# B&R Automation Studio project Y4_V3_1 (part 2)

### Acp10cfg.ncc - 5PPC2100_BY01_000/Motion/Acp10cfg.ncc
```
NcConfiguration (Version=2.46.0, NcSwId=Acp10)
  ACP10CF1_typ:
    cnt_nettrc_rec_drive = 150
    bufsize_trace_upload = 1200
    tc_nc_man_task = Cyclic #1
    glob_pv_as_ncobject = Yes
    ncsys_dl_broadcast = Yes
    ncsys_dl_acp_reset = Yes
    safemc_log_err_to_ax = Yes
    network_init:
      ncsw_init_execute = Yes
      automatic_execute = No
      node_nr_warning = Yes
      net_err_before_ncact = Yes
    nettrc:
      enter_parsecrec = Yes
      enter_ncaction = Yes
      save_ring_startidx = Yes
    cam_prof_download:
      cam_dat_dl_parallel = No
      tc_cam_dl_parallel = Task class for NC Manager task
    plk_if[0]:
      if_name = SL1.IF1
      tc_CycDat_PLCopen = Task class for NC Manager task
      mc_broadcast_extdat = No
    plk_if[1]:
      if_name = SS1.SS1.SS1.SS1.SS1
      tc_CycDat_PLCopen = Task class for NC Manager task
      mc_broadcast_extdat = No
    sdc_if[0]:
      if_name = SDC_IF1
      mc_broadcast_size = 800
      mc_broadcast_extdat = No
```

### Acp10map.ncm - 5PPC2100_BY01_000/Motion/Acp10map.ncm
```
NcMapping (NcSwId=Acp10, DisabledNodesAreHidden=False)
  NcObject Axis1 (ModuleId=8V1045.00-2a, Type=ncAXIS, Channel=1, AcoposSimulation=Off, InitParameter=axis1, AcoposParameter=table_par1, Disabled=FALSE, ModuleDisabled=FALSE)
  NcObject 8V1045.00-2a_ncV_AXIS1 (ModuleId=8V1045.00-2a, Type=ncV_AXIS, Channel=1, Disabled=TRUE, ModuleDisabled=FALSE)
  NcObject Axis2 (ModuleId=8V1045.00-2, Type=ncAXIS, Channel=1, AcoposSimulation=Off, InitParameter=axis1, AcoposParameter=table_par1, Disabled=FALSE, ModuleDisabled=FALSE)
  NcObject 8V1045.00-2_ncV_AXIS1 (ModuleId=8V1045.00-2, Type=ncV_AXIS, Channel=1, Disabled=TRUE, ModuleDisabled=FALSE)
  NcObject 8I74xxxxxxx.01P-1_ncAXIS1 (ModuleId=INV2, Type=ncAXIS, Channel=1, AcoposSimulation=Off, Disabled=TRUE, ModuleDisabled=FALSE)
  NcObject 8I74xxxxxxx.01P-1_ncAXIS1 (ModuleId=INV7, Type=ncAXIS, Channel=1, AcoposSimulation=Off, Disabled=TRUE, ModuleDisabled=FALSE)
  NcObject 8I74xxxxxxx.01P-1_ncAXIS1 (ModuleId=INV10, Type=ncAXIS, Channel=1, AcoposSimulation=Off, Disabled=TRUE, ModuleDisabled=FALSE)
  NcObject 8I74xxxxxxx.01P-1_ncAXIS1 (ModuleId=INV13, Type=ncAXIS, Channel=1, AcoposSimulation=Off, Disabled=TRUE, ModuleDisabled=FALSE)
  NcObject 8I74xxxxxxx.01P-1_ncAXIS1 (ModuleId=INV11, Type=ncAXIS, Channel=1, AcoposSimulation=Off, Disabled=TRUE, ModuleDisabled=FALSE)
  NcObject 8I74xxxxxxx.01P-1_ncAXIS1 (ModuleId=INV12, Type=ncAXIS, Channel=1, AcoposSimulation=Off, Disabled=TRUE, ModuleDisabled=FALSE)
```

## Configuration Simulation

CPU , AutomationRuntime D4.24, Vc V4.26.0

### Task classes (Cpu.sw)
```
Cyclic#1 (cycle 500 us, tolerance 100000 us):
  IO <- System.IO.prg
  LineConfig <- System.LineConfig.prg
  SensorInpu <- System.SensorInput.prg
  Seam1Array <- Motion.Seam1Array.prg
  Seam2Array <- Motion.Seam2Array.prg
Cyclic#2 (cycle 200000 us, tolerance 10000000 us):
  ResetInv <- Automatic.ResetInv.prg
  AxBlocks <- Automatic.AxBlocks.prg
  ConLoad <- Automatic.ConLoad.prg
  ConSeam1 <- Automatic.ConSeam1.prg
  ConCorner <- Automatic.ConCorner.prg
  ConSeam2 <- Automatic.ConSeam2.prg
  ConBuffers <- Automatic.ConBuffers.prg
  ConRow <- Automatic.ConRow.prg
  ConBatch <- Automatic.ConBatch.prg
  Seaming <- Automatic.Seaming.prg
  Batching <- Automatic.Batching.prg
  Modes <- Automatic.Modes.prg
  FlipUpArms <- Automatic.FlipUpArms.prg
  Outputs <- Automatic.Outputs.prg
Cyclic#3 (cycle 500000 us, tolerance 10000000 us):
  Control <- System.Control.prg
  Seamers <- System.Seamers.prg
  Process <- System.Process.prg
Cyclic#4 (cycle 1000000 us, tolerance 10000000 us):
  IPConfig <- IPConfig.IPConfig.prg
  Filstar <- System.Filstar.prg
  Level <- VisControl.HMIControl.Level.prg
  Status <- VisControl.HMIControl.Status.prg
  Start <- VisControl.HMIControl.Start.prg
  ESRecover <- VisControl.HMIControl.ESRecover.prg
  Simulation <- VisControl.HMIControl.Simulation.prg
  Page10 <- VisControl.HMIControl.Page10.prg
  Page11 <- VisControl.HMIControl.Page11.prg
  Page12 <- VisControl.HMIControl.Page12.prg
  Page13 <- VisControl.HMIControl.Page13.prg
  Page14 <- VisControl.HMIControl.Page14.prg
  Page15 <- VisControl.HMIControl.Page15.prg
  Page16 <- VisControl.HMIControl.Page16.prg
  Page17 <- VisControl.HMIControl.Page17.prg
  Page18 <- VisControl.HMIControl.Page18.prg
  Page20 <- VisControl.HMIControl.Page20.prg
  EPLComms <- InvComms.EPLComms.prg
  BatchData <- VisControl.BatchDisp.BatchData.prg
VcDataObjects: HMIXGA <- HMIXGA.HMIXGA.dob, BatchP <- BatchDisplay.BatchP.dob
Binaries: verdana, vcpkat, vctcal, HMIXGA03, vcgclass, vcnet, HMIXGA01, vcpdsw, vccshape, arialbd, arialn, vccstr, trebuc, vccnum, vcrt, visvc, vccbar, vcbclass, vcalarm, vcctext, vcmgr, vccovl, HMIXGA02, vccalarm, vcpfar00, vcdsloc, vccbtn, vcdsint, vcchspot, arial, vccpwd, vcfile, vcpdvnc, vcshared, vccbmp, vcfntttf, vccddbox, vccpopup, SRVXGA01, SRVXGA02, SRVXGA03, SRVXGA, BatchP01, BatchP03, BatchP02, acp10cfg, Acp10map, ashwd, arconfig, asfw, sysconf, iomap, Acp10sys, vcchtml, vccurl, vcxml, vccdt, VisuTe01, VisuTe02, VisuTe03, vcctrend, vccslider, vccline
Libraries: AsIecCon, astime, standard, sys_lib, Runtime, brsystem, powerlnk, DataObj, asstring, dvframe, AxisCtrl, AsARCfg, IecCheck, LoopConR, Visapi, vcresman, Acp10man, Acp10par, NcGlobal, fileio, Acp10_MC, Lib_Ashton, asepl, AsMath, arsvcreg
```

### Hardware
```
PC_any : PC_any v1.1.0.0 (OrderNumber=PC)
  Connector IF3:
    Vnc1
    VncVcObjectName1 = HMIXGA
    VncKeyMappingFile1 = VC\PS2-Keyboard.dis
    VncAuthentication1 = 1
    VncPasswordViewOnly1 = 1234
    VncPasswordViewControl1 = 4046
    VncRefreshRate1 = 100
    Vnc2
    VncVcObjectName2 = BatchP
    VncKeyMappingFile2 = VC\PS2-Keyboard1.dis
    VncPortNumber2 = 5902
  ConfigurationID = N13_V1_0_Simulation
  PermanentPvSize = 4096
  VolatileGlobalPvSize = 327679
  CyclicObjects = 250
  BRObjects = 600
  SystemTick = 500
  Cyclic1Duration = 500
  Cyclic1Tolerance = 100000
  Cyclic1Input = 1
  Cyclic2Duration = 200000
  Cyclic2Tolerance = 10000000
  Cyclic3Duration = 500000
  Cyclic3Tolerance = 10000000
  Cyclic4Duration = 1000000
  Cyclic4Tolerance = 10000000
  Cyclic5Duration = 2000000
  Cyclic5Tolerance = 10000000
  Cyclic6Duration = 3000000
  Cyclic6Tolerance = 12000000
  Cyclic7Duration = 4000000
  Cyclic7Tolerance = 12000000
  Cyclic8Duration = 5000000
  Cyclic8Tolerance = 30000000
```

### Cpu.per - PC_any/Cpu.per
```iecst
(********************************************************************
 * COPYRIGHT --
 ********************************************************************
 * File: Cpu.per
 * Author: NickE
 * Created: April 2, 2015
 ********************************************************************
 * Declaration of permanent variables
 ********************************************************************)
VAR_CONFIG
	Ax1P AT %M0; (*Axis 1 permananent variables*)
	Ax2P AT %M60; (*Axis 2 permananent variables*)
	Grind1 AT %M120; (*Grinding data permanent variables*)
	Grind2 AT %M176; (*Grinding data permanent variables*)
	Data AT %M232; (*Runtime data permanent variables*)
	PresetSys AT %M264; (*System timer presets*)
	SysPerm AT %M344; (*Permanent system variables*)
	PresetSeam AT %M368; (*Auto running timer presets*)
	RowPerm AT %M472; (*Row building permanent variables*)
	LoadPerm AT %M488; (*Load building permanent variables*)
	ArmsPerm1 AT %M504; (*Flip up arms retained values*)
	ArmsPerm2 AT %M528; (*Flip up arms retained values*)
	ScalePerm AT %M552; (*Conveyor scaling constants*)
	InvPerms AT %M608; (*Inverter Permanent Variables*)
	Speeds AT %M724; (*Conveyor speeds*)
	AnalogPerm AT %M768; (* *)
	TrackDelayPT AT %M1104; (*Preset for timeout*)
	NozzlePerm AT %M1364; (* *)
	InterceptPT AT %M1372; (* *)
END_VAR
```

### Acp10cfg.ncc - PC_any/Motion/Acp10cfg.ncc
```
NcConfiguration (Version=2.45.1, NcSwId=Acp10)
  ACP10CF1_typ:
    cnt_nettrc_rec_drive = 150
    bufsize_trace_upload = 1200
    tc_nc_man_task = Cyclic #1
    glob_pv_as_ncobject = Yes
    ncsys_dl_broadcast = Yes
    ncsys_dl_acp_reset = Yes
    safemc_log_err_to_ax = Yes
    network_init:
      ncsw_init_execute = Yes
      automatic_execute = No
      node_nr_warning = Yes
      net_err_before_ncact = Yes
    nettrc:
      enter_parsecrec = Yes
      enter_ncaction = Yes
      save_ring_startidx = No
    cam_prof_download:
      cam_dat_dl_parallel = No
      tc_cam_dl_parallel = Task class for NC Manager task
```

## Logical view

Binary libraries used (declarations not repeated): Runtime, Operator, standard, sys_lib, brsystem, powerlnk, AsIecCon, astime, DataObj, asstring, dvframe, AsARCfg, LoopConR 2.72.0, Visapi, AsEPL, AsMath, Acp10man 2.50.1, Acp10par 2.50.1, NcGlobal 2.50.1, Acp10_MC 2.50.1

### Global.typ - Global data types
```iecst
(********************************************************************
 * COPYRIGHT --
 ********************************************************************
 * File: Global.typ
 * Author: NickE
 * Created: April 2, 2015
 ********************************************************************
 * Global data types of project N_Default
 ********************************************************************)

TYPE
	SizeData_enum :
		(
		SD_Idle := 0, (*Wait*)
		SD_WidthData := 1, (*Set Width Data*)
		SD_WidthACK := 2, (*Wait for acknowledgement that width data has been received*)
		SD_NotWidthACK := 3, (*Wait for acknowledge off, data has transmitted*)
		SD_LengthData := 4, (*Set Length Data*)
		SD_LengthACK := 5, (*Wait for acknowledgement that length data has been received*)
		SD_NotLengthACK := 6 (*Wait for acknowledge off, data has transmitted*)
		);
	SizeData_typ : 	STRUCT
		Sizes : ARRAY[0..11]OF BOOL; (*Bit array to pass data to AGV controller*)
		Sequence : SizeData_enum;
		CurrentWidth : UINT;
		CurrentLength : UINT;
		WidthMask : BOOL;
		LengthMask : BOOL;
	END_STRUCT;
	Measurement_typ : 	STRUCT
		Reset : BOOL;
		Runtime : Display_enum;
	END_STRUCT;
	Alarm_typ : 	STRUCT
		Control : USINT; (*Visu alarm control*)
		Group : USINT; (*Visu alarm control*)
		Alarm : USINT; (*Visu alarm control*)
		Priority : USINT; (*Visu alarm control*)
	END_STRUCT;
	ANALOGCAPTURE_typ : 	STRUCT
		CLB : ANALOGRECORD_typ;
	END_STRUCT;
	ANALOGPERMS_typ : 	STRUCT
		V1 : ANALOGPERM_typ;
		C1 : ANALOGPERM_typ;
		C2 : ANALOGPERM_typ;
	END_STRUCT;
	ANALOGPERM_typ : 	STRUCT
		ActAnalog : REAL;
		ActSpeed : REAL;
	END_STRUCT;
	ANALOGRECORD_typ : 	STRUCT
		RecordStart : BOOL;
		RecordConfirm : BOOL;
		SpeedDisp : REAL;
		DisplayRaw : UINT;
		DisplaySpeed : REAL;
		DisplayAnalog : REAL;
	END_STRUCT;
	ANALOGS_typ : 	STRUCT
		CL1 : ANALOGPERMS_typ;
		CS1 : ANALOGPERMS_typ;
		CV1 : ANALOGPERMS_typ;
		CC1 : ANALOGPERMS_typ;
		CC2 : ANALOGPERMS_typ;
		CS2 : ANALOGPERMS_typ;
		CV2 : ANALOGPERMS_typ;
		CC3 : ANALOGPERMS_typ;
		CC4 : ANALOGPERMS_typ;
		CB1 : ANALOGPERMS_typ;
		CB2 : ANALOGPERMS_typ;
		CRB : ANALOGPERMS_typ;
		CRE : ANALOGPERMS_typ;
		CLB : ANALOGPERMS_typ;
	END_STRUCT;
	ArmsPerm_typ : 	STRUCT
		Position : ARRAY[0..5]OF REAL; (*Position for operation comparison*)
	END_STRUCT;
	ArmsTemp_typ : 	STRUCT
		HoldUp : TrackCount; (*Count for arms hold up*)
		UpCheck : INT; (*Case statement index*)
		DownDone : BOOL; (*Done bit for all down condition*)
		UpDone : BOOL; (*Done bit for selected up comparison.*)
		Down : ARRAY[0..10]OF BOOL; (*Down comparison bits*)
		Up : ARRAY[0..10]OF BOOL; (*Up comparison bits*)
		ActPos : REAL; (*Actual Position*)
	END_STRUCT;
	AxisBasic_typ : 	STRUCT
		Power : BOOL; (*Turns the power on*)
		Home : BOOL; (*homes the axis*)
		MoveAbsolute : BOOL; (*Starts the absolute movement*)
		Stop : BOOL; (*Stops a movement*)
		MoveJogPos : BOOL; (*Starts the jog movement in positive direction*)
		MoveJogNeg : BOOL; (*Starts the jog movement in negative direction*)
		ErrorAcknowledge : BOOL; (*Acknowledge an error with a pos. Edge*)
		ParaPosition : REAL; (*Parameter absolute target position*)
		ParaVelocity : REAL; (*Parameter target velocity*)
		ParaDirection : USINT; (*Parameter movement direction*)
		ParaAcceleration : REAL; (* Parameter movement acceleration*)
		ParaDeceleration : REAL; (* Parameter movement deceleration*)
		ParaHomePosition : REAL; (*Parameter home position*)
		ParaJogVelocity : REAL; (*Parameter jog movement target velocity*)
		ParaOverrideVelocity : REAL; (*Parameter velocity override (0.0 - 2.0)*)
		ParaOverrideAcceleration : REAL; (*Parameter acceleration override (0.0001 - 2.0)*)
		ErrorID : UINT; (*Shows the Error ID (0 = No Error)*)
		ErrorText : ARRAY[0..3]OF STRING[79]; (*Shows the Acopos Errortext as string*)
		ActPosition : REAL; (*actual position*)
		ActVelocity : REAL; (*actual velocity*)
		StatusDisabled : BOOL; (*Status power disabled*)
		StatusStandstill : BOOL; (*Status axis at standstill*)
		StatusStopping : BOOL; (*Status axis is stopping*)
		StatusHoming : BOOL; (*Status axis is homing*)
		StatusMotionDiscrete : BOOL; (*Status discrete motion is active*)
		StatusMotionContinous : BOOL; (*Status continous motion is active*)
		StatusMotionSynchronized : BOOL; (*Status synchronized motion is active*)
		StatusErrorstop : BOOL; (*Status axis stopped after error*)
		Obj : UDINT; (*Pointer to NC structure*)
		Step : USINT; (*State index*)
		ErrorNcAccess : UINT; (*ncaccess function status*)
		CyclicBits : UDINT; (*Cyclic read data address*)
		StartHome : BOOL; (*Start homing*)
		Homed : BOOL; (*Homing done*)
		Ret : UDINT; (*memcpy status*)
		CyclicReadExecute : BOOL; (*Execute cyclic read*)
		OKtoRun : BOOL; (*Cyclic read completed*)
		DigiSetup : BOOL; (*Map X67 inputs to ACOPOS*)
	END_STRUCT;
	AxisPerm_typ : 	STRUCT
		FastSpeed : REAL; (*Fast search velocity*)
		SlowSpeed : REAL; (*Slow search velocity*)
		FCSpeed : REAL; (*Forward check search speed*)
		FwdFeed : REAL; (*Forward feed length*)
		RevFeed : REAL; (*Reverse feed length*)
		AbsMax : REAL; (*Maximum absolute position*)
		AbsMin : REAL; (*Minimum absolute position*)
		FFAbsMax : REAL; (*Fast forward absolute position*)
		FRAbsMin : REAL; (*Fast rev absolute position*)
		FCDist : REAL; (*Forward check distance*)
		SlowAdj1 : REAL; (*Reverse slow adjustment*)
		SlowAdj2 : REAL; (*Forward slow adjustment*)
		SlowAdj3 : REAL; (*Forward check adjustment*)
		SlowDist : REAL; (*Slow move distance*)
		Origin : REAL; (*Origin Preset Position*)
	END_STRUCT;
	AXIS_STATE_enum :
		(
		STATE_DIGI_SETUP := 0, (*constant for mapping PL inputs to ACOPOS*)
		STATE_WAIT := 1, (*constant for a waiting step*)
		STATE_POWER_ON := 2, (*constant for the step in which the controller is switched on*)
		STATE_HOME := 3, (*constant for the step in which the axis is homed*)
		STATE_READY := 10, (*constant for a waiting step*)
		STATE_STOP := 11, (*constant for the step in which movements are stopped*)
		STATE_MOVE_ABSOLUTE := 14, (*constant for the step in which a movement to defined position is started*)
		STATE_JOG_POSITIVE := 12, (*constant for the step in which a positive jogging movement is executed*)
		STATE_JOG_NEGATIVE := 13, (*constant for the step in which a negative jogging movement is executed*)
		STATE_MOVE_ADDITIVE := 15, (*constant for the step in which a movement with defiened distance is started*)
		STATE_MOVE_VELOCITY := 16, (*constant for the step in which a movement with defined velocity is started*)
		STATE_HALT := 17, (*constant for the step in which movements are stopped*)
		STATE_ERROR_AXIS := 100, (*constant for the axis error step*)
		STATE_ERROR := 101, (*constant for the error step*)
		STATE_ERROR_RESET := 102 (*constant for the step in which the errors are reset*)
		);
	Axis_typ : 	STRUCT
		CheckPosition : REAL; (*Absolute move start position*)
		Error : BOOL; (*Axis error*)
		OriginSet : BOOL; (*Origin search complete*)
		Reset : BOOL; (*Reset after error*)
		SeekFin : BOOL; (*Seek and find complete*)
		Seek1 : BOOL; (*Start seek and find*)
		Seek1Disp : USINT; (*Runtime control*)
		Seek2 : BOOL; (*Restart seek and find*)
		Count : USINT; (*Seek and find completion count*)
		Measure : REAL; (*Final stop position*)
		Pattern : PATTERN_enum; (*Seek and find case control*)
		ResetEnable : Status_enum := HIDE; (*Enable reset button for Visu*)
		Sensors : USINT; (*Seek and find sensor array status*)
		Text : USINT; (*Seek and find status*)
		Max : Limit_typ; (*Maximum limits*)
		Min : Limit_typ; (*Minimum limits*)
		Block : BOOL; (*Block axis movement*)
		Blocks : ARRAY[0..12]OF BOOL; (*Block conditions*)
		HiVol : BOOL; (*High Volume Latch*)
		RaiseArms : BOOL; (*On only when arms to be raised*)
		Active : BOOL; (*On only when seek and find to be active*)
		Seek2Runtime : USINT; (*Runtime control for manual seek and find*)
		MovetoPosition : REAL; (*Optimisation position to move to*)
		StartCheck : BOOL; (*Check Move Started*)
		Node : STRING[49]; (*Module address for motion limits*)
	END_STRUCT;
	basic_axisState_typ : 	STRUCT  (*axis state structure*)
		Disabled : BOOL; (*if set, axis is in state Disabled*)
		StandStill : BOOL; (*if set, axis is in state StandsStill*)
		Homing : BOOL; (*if set, axis is in state Homing*)
		Stopping : BOOL; (*if set, axis is in state Stopping*)
		DiscreteMotion : BOOL; (*if set, axis is in state DiscreteMotion*)
		ContinuousMotion : BOOL; (*if set, axis is in state ContinousMotion*)
		SynchronizedMotion : BOOL; (*if set, axis is in state SynchronizedMotion*)
		ErrorStop : BOOL; (*if set, axis is in state ErrorStop*)
	END_STRUCT;
	basic_command_typ : 	STRUCT  (*command structure*)
		Obj : UDINT; (*axis reference*)
		Step : AXIS_STATE_enum; (*current step in the step sequence*)
		Power : BOOL; (*switch on the controller*)
		Home : BOOL; (*reference the axis*)
		MoveAbsolute : BOOL; (*move to an defined position*)
		MoveAdditive : BOOL; (*move a defiened distance*)
		MoveVelocity : BOOL; (*start a movement with a defiened velocity*)
		Halt : BOOL; (*stop every active movement*)
		Stop : BOOL; (*stop every active movement as long as is set*)
		MoveJogPos : BOOL; (*move in positive direction as long as is set*)
		MoveJogNeg : BOOL; (*move in negative direction as long as is set*)
		ErrorAcknowledge : BOOL; (*reset active errors*)
	END_STRUCT;
	basic_parameter_typ : 	STRUCT  (*parameter structure*)
		Position : REAL; (*target-position for MoveAbsolute-Command*)
		Distance : REAL; (*distance for MoveAdditive-Command*)
		Velocity : REAL; (*velocity for MoveVelocity-Command*)
		Direction : USINT; (*direction for commanded movements*)
		Acceleration : REAL; (*acceleration for commanded movements*)
		Deceleration : REAL; (*deceleration for commanded movements*)
		HomePosition : REAL; (*target-position for referencing the axis*)
		HomeMode : USINT; (*homing mode*)
		JogVelocity : REAL; (*velocity for jogging movement*)
	END_STRUCT;
	basic_status_typ : 	STRUCT  (*status structure*)
		ErrorID : UINT; (*ErrorID of any occured error*)
		ErrorText : ARRAY[0..3]OF STRING[79]; (*Error Text*)
		ActPosition : REAL; (*actual position of the axis*)
		ActVelocity : REAL; (*actual velocity of the axis*)
		DriveStatus : MC_DRIVESTATUS_TYP; (*actual status of the axis*)
	END_STRUCT;
	basic_typ : 	STRUCT  (*control structure*)
		Command : basic_command_typ; (*command structure*)
		Parameter : basic_parameter_typ; (*parameter structure*)
		Status : basic_status_typ; (*status structure*)
		AxisState : basic_axisState_typ; (*axis state structure*)
	END_STRUCT;
	BeltClear_typ : 	STRUCT
		NonProcess1 : BOOL; (*Non additional process belt 1*)
		NonProcess2 : BOOL; (*Non additional process belt 2*)
		Process1 : BOOL; (*Additional process belt 1*)
		Process2 : BOOL; (*Additional process belt 2*)
		Start : BOOL; (*Start latch*)
		Done : BOOL; (*Clear of Belts*)
	END_STRUCT;
	DataFlow_typ : 	STRUCT
		IndexRow : USINT;
		IndexLoad : USINT;
	END_STRUCT;
	EMO_typ : 	STRUCT
		Confirm : ARRAY[0..4]OF BOOL; (*Visu control*)
		Disp : ARRAY[0..4]OF Status_enum; (*Visu control*)
		Latch1 : BOOL; (*Latch to block conveyor movement*)
		Latch2 : BOOL; (*Latch to block conveyor movement*)
		Latch3 : BOOL; (*Latch to block conveyor movement*)
		Latch4 : BOOL; (*Latch to block conveyor movement*)
		LatchTON1 : TON; (*EMO finish delay timer*)
		LatchTON2 : TON; (*EMO finish delay timer*)
		LatchTON3 : TON; (*EMO finish delay timer*)
		LatchTON4 : TON; (*EMO finish delay timer*)
		Recovery : BOOL; (*During recovery sequence*)
		Start : TON; (*EMO start delay timer*)
		StartLatch : BOOL; (*Latch condition after EMO*)
	END_STRUCT;
	EPLState_typ : 	STRUCT
		LinkOK : BOOL;
		CycleOK : BOOL;
		SyncOK : BOOL;
	END_STRUCT;
	Filstar_typ : 	STRUCT
		Out : BOOL; (*Valve output*)
		Open : TON; (*Valve open delay*)
		Interval : TON; (*Interval delay*)
	END_STRUCT;
	GrindDisp_typ : 	STRUCT
		ShiftDisp : Status_enum; (*Visu control*)
		TotalDisp : Status_enum; (*Visu control*)
	END_STRUCT;
	Grind_typ : 	STRUCT
		ShiftMs : UINT; (*Milliseconds ground 0-999*)
		ShiftSec : UINT; (*Seconds ground 0-59*)
		ShiftMin : UINT; (*Minutes ground 0-59*)
		ShiftHr : UINT; (*Hours ground 0-23*)
		ShiftDay : UINT; (*Days ground*)
		ShiftFtLow : UDINT; (*Length ground feet lower 9 digits*)
		ShiftFtUpp : UDINT; (*Length ground feet upper 9 digits*)
		ShiftMLow : UDINT; (*Length ground metres lower 9 digits*)
		ShiftMUpp : UDINT; (*Length ground metres upper 9 digits*)
		TotalMs : UINT; (*Milliseconds ground 0-999*)
		TotalSec : UINT; (*Seconds ground 0-59*)
		TotalMin : UINT; (*Minutes ground 0-59*)
		TotalHr : UINT; (*Hours ground 0-23*)
		TotalDay : UINT; (*Days ground*)
		TotalFtLow : UDINT; (*Length ground feet lower 9 digits*)
		TotalFtUpp : UDINT; (*Length ground feet upper 9 digits*)
		TotalMLow : UDINT; (*Length ground metres lower 9 digits*)
		TotalMUpp : UDINT; (*Length ground metres upper 9 digits*)
	END_STRUCT;
	Input_typ : 	STRUCT
		In : BOOL; (*Input bit*)
		Int : BOOL; (*Internal bit*)
		Latch : BOOL; (*Latch for start of track steps where sensor not present*)
		BlockDisp : Status_enum; (*Display warning when blocking following glass*)
	END_STRUCT;
	InvPerms_typ : 	STRUCT
		CL1 : InvPerm_typ; (*Inverter saved parameters*)
		CS1 : InvPerm_typ; (*Inverter saved parameters*)
		CV1 : InvPerm_typ; (*Inverter saved parameters*)
		CC1 : InvPerm_typ; (*Inverter saved parameters*)
		CC2 : InvPerm_typ; (*Inverter saved parameters*)
		CS2 : InvPerm_typ; (*Inverter saved parameters*)
		CV2 : InvPerm_typ; (*Inverter saved parameters*)
		CC3 : InvPerm_typ; (*Inverter saved parameters*)
		CC4 : InvPerm_typ; (*Inverter saved parameters*)
		CB1 : InvPerm_typ; (*Inverter saved parameters*)
		CB2 : InvPerm_typ; (*Inverter saved parameters*)
		CRB : InvPerm_typ; (*Inverter saved parameters*)
		CRE : InvPerm_typ; (*Inverter saved parameters*)
		CLB : InvPerm_typ; (*Inverter saved parameters*)
		SetValues : BOOL;
	END_STRUCT;
	InvPerm_typ : 	STRUCT
		Accel : UINT; (*Value for ACC, Acceleration*)
		Decel : UINT; (*Value for DEC, Deceleration*)
		Analog : FB_ANALOG_enum; (*Analog type selection*)
	END_STRUCT;
	LegTest_enum :
		(
		TEST_OFF := 0,
		TEST_ON_STOP := 1,
		TEST_LEG1 := 2,
		TEST_LEG2 := 3,
		TEST_LEG3 := 4,
		TEST_LEG4 := 5
		);
	LegTest_typ : 	STRUCT
		Disp : Status_enum := HIDE; (*Runtime control*)
		Index : LegTest_enum := TEST_OFF; (*Case Index*)
	END_STRUCT;
	Limit_typ : 	STRUCT
		UppO : REAL; (*Upper limit for visu input*)
		UppF : REAL; (*Upper limit for visu input*)
		Upp : REAL; (*Upper limit for visu input*)
		LowO : REAL; (*Lower limit for visu input*)
		LowF : REAL; (*Lower limit for visu input*)
		Low : REAL; (*Lower limit for visu input*)
	END_STRUCT;
	LoadPerm_typ : 	STRUCT
		FurnClear : UDINT; (*Type of Furnace clear signal, Pulse or On.*)
		Max : REAL; (*Maximum batch length*)
		Gap : REAL; (*Actual gap*)
		ClearPT : UDINT; (*Preset time for manual batch clear*)
	END_STRUCT;
	Machine : 	STRUCT
		ErrorText : ARRAY[0..3]OF STRING[79];
		ErrorID : UINT;
		ErrorAcknowledge : BOOL;
		JogNegative : BOOL;
		JogPositive : BOOL;
		Stop : BOOL;
		Start : BOOL;
		MasterStop : BOOL;
		Mode : BOOL;
		Power : BOOL;
	END_STRUCT;
	Mode_typ : 	STRUCT
		Count : TrackCount; (*Count tracking bits*)
		Clear1 : TON; (*Delay before clear*)
		Clear2 : TON; (*Delay before clear*)
		Clear : BOOL; (*EMO Clear*)
		Input1 : BOOL; (*Mode selection*)
		Input2 : BOOL; (*Mode selection*)
		Input3 : BOOL; (*Mode selection*)
		Input4 : BOOL; (*Mode selection*)
		Active : BOOL; (*Mode active*)
		Clearing : BOOL; (*Mode clearing*)
		ESDisp : USINT; (*Visu display control*)
		Disp : Status_enum := HIDE; (*Visu display control*)
		Selected : BOOL; (*Mode selected but not active.*)
		Blocked : BOOL; (*Block preceding systems*)
	END_STRUCT;
	Output_typ : 	STRUCT
		Auto : BOOL; (*Output during auto operation*)
		Test : BOOL; (*Output during test operation*)
		Trip : BOOL; (*Linked trip input*)
		PalUp : BOOL; (*Pallet Up at EStop*)
		PalDown : BOOL; (*Pallet Down at EStop*)
	END_STRUCT;
	PATTERN_enum :
		(
		READY := 0, (*Ready to start Search Pattern*)
		FAST_REV := 1, (*Fast Reverse Search Pattern*)
		SLOW_REV := 2, (*Slow Reverse Search Pattern*)
		CHECK := 3, (*Verify Stop Position Search Pattern*)
		SLOW_FWD := 4, (*Slow Forward Search Pattern*)
		FAST_FWD := 5 (*Fast Forward Search Pattern*)
		);
	PermSys_typ : 	STRUCT
		PasswordDefault : BOOL; (*Reset passwords to default*)
		Password : ARRAY[0..3]OF STRING[4]; (*Password storage*)
	END_STRUCT;
	Perms_typ : 	STRUCT
		FurnReady : USINT;
		HiVolume : STATE_enum;
		VersionText : STRING[30]; (*Version Text*)
		FLIPARMS1 : SINT; (*Seamer 1 No of Flip Up arms*)
		FLIPARMS2 : SINT; (*Seamer 2 No of Flip Up arms*)
	END_STRUCT;
	PLInvOut_typ : 	STRUCT
		Fast : ARRAY[0..5]OF BOOL := [6(FALSE)]; (*Multiple start conditions ??Is this needed. Just change speed reference*)
		Run : ARRAY[0..5]OF BOOL := [6(FALSE)]; (*Multiple start conditions*)
		Rev : ARRAY[0..5]OF BOOL := [6(FALSE)]; (*Multiple start conditions*)
		Slow : ARRAY[0..5]OF BOOL := [6(FALSE)]; (*Multiple start conditions ??Is this needed. Just change speed reference*)
		Blower : BOOL := FALSE; (*Overblower*)
		SpeedRef : REAL; (*Speed Reference (Hz)*)
	END_STRUCT;
	PLInvScale_typ : 	STRUCT
		CL1Scale : REAL; (*Speed scaling CL1*)
		CS1Scale : REAL; (*Speed scaling CS1*)
		CV1Scale : REAL; (*Speed scaling CV1*)
		CC1Scale : REAL; (*Speed scaling CC1*)
		CC2Scale : REAL; (*Speed scaling CC2*)
		CS2Scale : REAL; (*Speed scaling CS2*)
		CV2Scale : REAL; (*Speed scaling CV2*)
		CC3Scale : REAL; (*Speed scaling CC3*)
		CC4Scale : REAL; (*Speed scaling CC4*)
		CB1Scale : REAL; (*Speed scaling CB1*)
		CB2Scale : REAL; (*Speed scaling CB2*)
		CRBScale : REAL; (*Speed scaling CRB*)
		CREScale : REAL; (*Speed scaling CRE*)
		CLBScale : REAL; (*Speed scaling CLB*)
	END_STRUCT;
	PLINV_In_typ : 	STRUCT
		ETAD_00 : BOOL; (*Status parameter (1 = Ready to switch on, awaiting power section line supply)*)
		ETAD_01 : BOOL; (*Status parameter (1 = Switched on, ready)*)
		ETAD_02 : BOOL; (*Status parameter (1 = Operation enabled, running)*)
		Fault : BOOL; (*Status parameter (1 = Fault detection) ETAD_03*)
		ETAD_04 : BOOL; (*Status parameter (1= Voltage enabled, power section line supply present)*)
		ETAD_05 : BOOL; (*Status parameter (0 = Quick stop, emergency stop)*)
		ETAD_06 : BOOL; (*Status parameter (1 = Switch on disabled, power section line supply disabled)*)
		ETAD_07 : BOOL; (*Status parameter (1 = Warning, alarm)*)
		ETAD_09 : BOOL; (*Status parameter (0 = Command or reference via terminals; 1 = Command or reference via network)*)
		ETAD_10 : BOOL; (*Status parameter (1 = Target reached, reference reached)*)
		ETAD_11 : BOOL; (*Status parameter (1 = Internal limit active, reference outside limits)*)
		ETAD_14 : BOOL; (*Status parameter (1 = STOP via stop key)*)
		ETAD_15 : BOOL; (*Status parameter (Direction of rotation 0 = Forward rotation; 1 = Reverse rotation)*)
		HMIS : UINT; (*Drive state*)
		ETI_00 : BOOL; (*Extended status word (1 = Access to the EEPROM non-volatile memory in progress)*)
		ETI_01 : BOOL; (*Extended status word (0 = No parameter consistency check; 1 = Parameter consistency check)*)
		ETI_02 : BOOL; (*Extended status word (0 = The drive is not in fault state or a fault is detected; 1 = The drive is in fault state but the fault is no longer present (not reset))*)
		ETI_04 : BOOL; (*Extended status word (1 = The drive is in speed mode)*)
		ETI_05 : BOOL; (*Extended status word (1 = DC injection)*)
		ETI_06 : BOOL; (*Extended status word (0 = Drive in steady state; 1 = Drive in transient state)*)
		ETI_07 : BOOL; (*Extended status word (1 = Motor thermal state threshold reached for the active motor)*)
		ETI_08 : BOOL; (*Extended status word (1 = Overbraking)*)
		ETI_09 : BOOL; (*Extended status word (1 = Acceleration in progress)*)
		ETI_10 : BOOL; (*Extended status word (1 = Deceleration in progress)*)
		ETI_11 : BOOL; (*Extended status word (1 = Current limit in progress)*)
		ETI_12 : BOOL; (*Extended status word (1 = Fast stop in progress)*)
		ETI_13 : BOOL; (*Extended status word (bit 13 = 0 and bit 14 = 0 : Drive controled by terminal or local keypad; bit 13 = 1 and bit 14 = 0 : Drive controled by remote keypad; bit 13 = 0 and bit 14 = 1 : Drive controled by Modbus; bit 13 = 1 and bit 14 = 1 : Reserved)*)
		ETI_14 : BOOL; (*Extended status word (bit 13 = 0 and bit 14 = 0 : Drive controled by terminal or local keypad; bit 13 = 1 and bit 14 = 0 : Drive controled by remote keypad; bit 13 = 0 and bit 14 = 1 : Drive controled by Modbus; bit 13 = 1 and bit 14 = 1 : Reserved)*)
		ETI_15 : BOOL; (*Extended status word (0 = Forward operation applied before the ramp; 1 = Reverse operation applied before the ramp)*)
		RFR : INT; (*Output frequency [Hz] (Range depends on CMI_Output_Bool_09)*)
		OTR : INT; (*Motor torque (with filter) [0.1 %]*)
		LCR : UINT; (*Motor current (with filter) [0.1 A]*)
		THD : UINT; (*Drive thermal state [%]*)
		THR : UINT; (*Motor thermal state [%]*)
		ULN : UINT; (*Mains voltage [0.1 V]*)
		UOP : UINT; (*Motor voltage [1 V]*)
		IL1R_00 : BOOL; (*Logic input state (Value of LI1)*)
		IL1R_01 : BOOL; (*Logic input state (Value of LI2)*)
		IL1R_02 : BOOL; (*Logic input state (Value of LI3)*)
		IL1R_03 : BOOL; (*Logic input state (Value of LI4)*)
		IL1R_04 : BOOL; (*Logic input state (Value of LI5)*)
		IL1R_05 : BOOL; (*Logic input state (Value of LI6)*)
		OL1R_01 : BOOL; (*Relay 01 state*)
		OL1R_02 : BOOL; (*Relay 02 state*)
		OL1R_09 : BOOL; (*Logic output state*)
		AI1R : INT; (*Analog input 1 standardized value (+/- 8192)*)
		AI2R : INT; (*Analog input 2 standardized value (0 to 8192)*)
		AI3R : INT; (*Analog input 3 standardized value (0 to 8192)*)
		ERRD : UINT; (*CiA402 fault code*)
		LFT : INT; (*Last detected fault*)
		FNB : UINT; (*Fault counter*)
		STOS : UINT; (*STO status*)
		SLSS : UINT; (*SLS status*)
		SS1S : UINT; (*SS1 status*)
	END_STRUCT;
	PLINV_Out_typ : 	STRUCT
		CMDD_00 : BOOL; (*Control word (1 = Switch on)*)
		CMDD_01 : BOOL; (*Control word (0 = Disable voltage)*)
		CMDD_02 : BOOL; (*Control word (0 = Quick stop/Emergency stop)*)
		CMDD_03 : BOOL; (*Control word (1 = Enable operation/Run command)*)
		CMDD_07 : BOOL; (*Control word (Fault reset/Fault acknowledgment active on 0 -> 1 rising edge)*)
		CMDD_08 : BOOL; (*Control word (0 = RUN asked; 1 = STOP asked)*)
		CMDD_11 : BOOL; (*Control word (Direction of rotation 0 = Forward rotation; 1 = Reverse rotation)*)
		CMDD_12 : BOOL; (*Can be assigned to a command*)
		CMDD_13 : BOOL; (*Can be assigned to a command*)
		CMDD_14 : BOOL; (*Can be assigned to a command*)
		CMDD_15 : BOOL; (*Can be assigned to a command*)
		CMI_00 : BOOL; (*Extended control word (Factory setting command active at 1)*)
		CMI_01 : BOOL; (*Extended control word (Save configuration to EEPROM non-volatile memory command active at 1)*)
		CMI_02 : BOOL; (*Extended control word (Restore configuration to EEPROM non-volatile memory command active on 0 -> 1 rising edge)*)
		CMI_09 : BOOL; (*Extended control word Definition of the frequency reference (LFr) and output frequency (rFr) unit (0 = 0.1 Hz;  1 = Standardized value 16 signed bits based on the maximum frequency)*)
		CMI_15 : BOOL; (*Extended control word (Parameter consistency check 0 = check is activated; 1 = check is deactivated)*)
		LFR : INT; (*Frequency setpoint [Hz] (Range depends on CMI_Output_Bool_09)*)
		OL1R_01 : BOOL; (*Relay 01*)
		OL1R_02 : BOOL; (*Relay 02*)
		OL1R_09 : BOOL; (*Logic output 01*)
		AO1R : INT; (*Analog output 1 standardized value (0 to 8192)*)
	END_STRUCT;
	PLINV_typ : 	STRUCT
		Input : PLINV_In_typ; (*Input from Inverter*)
		Output : PLINV_Out_typ; (*Output to Inverter*)
		Inv : PLInv_typ; (*Control*)
		Brake : BOOL; (*Brake Output*)
		Reset : BOOL; (*Confirm reset from HMI*)
		o : PLInvOut_typ; (*Output Values*)
		Module : PLModule_typ; (*Module Information*)
		LastSpeed : REAL := 10.0; (*Last used speed*)
		SpeedAnalog : REAL; (*Speed value generated by analog value*)
	END_STRUCT;
	PLInv_typ : 	STRUCT
		Reference1 : ARRAY[0..1]OF lcrCurveByPoints_TabEntry_type; (*Frequency conversion reference points*)
		Scale1 : LCRCurveByPoints; (*M/Min to Frequency conversion table.*)
		SpeedTest : REAL := 15.0; (*Test Speed (m/min)*)
		Test : USINT; (*Visu Test Control*)
	END_STRUCT;
	Loads_typ : 	STRUCT
		Empty : RecordRows_typ;
		AshtonExit : RecordRows_typ;
		Furnace1 : RecordRows_typ;
		Furnace2 : RecordRows_typ;
		Furnace3 : RecordRows_typ;
		Furnace4 : RecordRows_typ;
		Furnace5 : RecordRows_typ;
		Furnace6 : RecordRows_typ;
		Furnace7 : RecordRows_typ;
		Furnace8 : RecordRows_typ;
		Furnace9 : RecordRows_typ;
		FurnaceExit : RecordRows_typ;
	END_STRUCT;
	PLModule_typ : 	STRUCT
		OK : BOOL; (*Module status (1 = module present)*)
		SerialNumber : UDINT; (*Serial Number*)
		ID : UDINT; (*Module ID*)
		HardwareVariant : UDINT; (*Hardware variant*)
		FirmwareVersion : UDINT; (*Firmware version*)
		ID_ACPi : UDINT; (*PL Module ID*)
		SerialNumber_ACPi : UDINT; (*PL Serial Number*)
	END_STRUCT;
	Preset_typ : 	STRUCT
		Buzzer : UDINT; (*Buzzer duration*)
		ESRestart : ARRAY[0..4]OF UDINT; (*Seamer conveyor delay during EMO recovery*)
		Filstar : ARRAY[0..2]OF UDINT; (*Filstar delays*)
		Belt : UDINT; (*During Belt auto start*)
		Extraction : UDINT; (*During Extraction auto start*)
		ED : UDINT; (*During ED auto start*)
		Vac : UDINT; (*During Vacuum auto start*)
		Water : ARRAY[0..4]OF UDINT; (*Water Pump delays*)
		Standby : UDINT; (*Before system standby*)
		VacsStop : UDINT; (*Vacuum run on after control stop*)
	END_STRUCT;
	Process_typ : 	STRUCT
		ShiftPiece : LREAL; (*Piece count*)
		ShiftMins : UINT; (*Runtime minutes*)
		ShiftHrs : UINT; (*Runtime hours*)
		ShiftDays : UINT; (*Runtime days*)
		ShiftYrs : UINT; (*Runtime years*)
		TotalPiece : LREAL; (*Piece count*)
		TotalMins : UINT; (*Runtime minutes*)
		TotalHrs : UINT; (*Runtime hours*)
		TotalDays : UINT; (*Runtime days*)
		TotalYrs : UINT; (*Runtime years*)
	END_STRUCT;
	Imperialification_typ : 	STRUCT
		WholeInchREAL : REAL;
		WholeInch : INT;
		Remainder : REAL;
		SixteenthStr : STRING[6];
		Sixteenth : REAL;
		float_len : UINT;
	END_STRUCT;
	PTCon_typ : 	STRUCT
		Slow : UDINT; (*Slow before stop or reverse*)
		Start : UDINT; (*Before start*)
		Clear : UDINT; (*Before clear*)
		Rev : UDINT; (*Reverse before stop*)
	END_STRUCT;
	PTSeam_typ : 	STRUCT
		BeltOn : ARRAY[0..12]OF UDINT; (*Delay before belt solenoid on*)
		BeltOff : ARRAY[0..12]OF UDINT; (*Delay before belt solenoid off*)
	END_STRUCT;
	RecordRows_typ : 	STRUCT
		Rows : ARRAY[0..15]OF RecordRow_typ;
		NotEmpty : BOOL;
	END_STRUCT;
	RecordRow_typ : 	STRUCT
		Row : ARRAY[0..12]OF Record_typ;
		NotEmpty : BOOL;
	END_STRUCT;
	Record_typ : 	STRUCT
		Width : REAL;
		Length : REAL;
	END_STRUCT;
	Reset_typ : 	STRUCT
		Grind : BOOL; (*Shift grind reset*)
		Time : BOOL; (*Shift time reset*)
		Count : BOOL; (*Shift count reset*)
		Total : BOOL; (*Total reset*)
	END_STRUCT;
	RowPerm_typ : 	STRUCT
		CenterDist : REAL; (*Centering distance*)
		CenterSpeed : REAL; (*Centering speed*)
		Max : REAL; (*Maximum row size*)
		Gap : REAL; (*Actual gap*)
	END_STRUCT;
	Rows_typ : 	STRUCT
		Empty : RecordRow_typ;
		Tracking30 : RecordRow_typ;
		Tracking40 : RecordRow_typ;
		Tracking41 : RecordRow_typ;
		Tracking50 : RecordRow_typ;
	END_STRUCT;
	Seamer_typ : 	STRUCT
		Stop1 : BOOL; (*Initiate Belt Off Delays Seamer 1*)
		Stop2 : BOOL; (*Initiate Belt Off Delays Seamer 2*)
		Start1 : BOOL; (*Initiate Belt On Delays Seamer 1*)
		Start2 : BOOL; (*Initiate Belt On Delays Seamer 2*)
	END_STRUCT;
	Simulation_typ : 	STRUCT
		On : BOOL; (*Simulation ON*)
		Disp : Status_enum := HIDE; (*Display for visu*)
	END_STRUCT;
	Warnings_typ : 	STRUCT
		AckDisp : Status_enum := HIDE; (*Display acknowledge warning*)
		Ack : BOOL; (*Acknowledge warning from visu*)
		Block : BOOL; (*Disable warnings*)
		Button : Status_enum := HIDE; (*Display warning button*)
		Delay : ARRAY[0..50]OF TON; (*Delays for timeouts*)
		Timeout : ARRAY[0..50]OF BOOL; (*Timeout active*)
		Acks : ARRAY[0..50]OF BOOL; (*Timeout not acknowledged*)
		Warningi : USINT; (*Array index*)
		i : USINT; (*Array index*)
		BlockTemp : BOOL; (*On at EMO.Latch**)
		iMax : USINT := 50; (*Array Index Max value*)
	END_STRUCT;
	STATE_enum :
		(
		OFF := 0,
		ON := 1,
		NO := 2,
		YES := 3
		);
	Status_enum :
		(
		SHOW := 0, (*Control visible with input enabled*)
		HIDE := 1, (*Control hidden*)
		LOCK := 2 (*Control visible with input disabled*)
		);
	TempSys_typ : 	STRUCT
		Alarm : BOOL; (*Configured alarm on*)
		Alarms : ARRAY[0..80]OF BOOL; (*Active alarms*)
		Alarmi : USINT; (*Array index*)
		Events : ARRAY[0..99]OF BOOL; (*Events*)
		Warning : BOOL; (*Configured warning on*)
		Warningi : USINT; (*Array index*)
	END_STRUCT;
	TrackDelayPT_typ : 	STRUCT
		PTTrack001 : UDINT; (*Track Delay preset*)
		PTTrack002 : UDINT; (*Track Delay preset*)
		PTTrack003 : UDINT; (*Track Delay preset*)
		PTTrack004 : UDINT; (*Track Delay preset*)
		PTTrack005 : UDINT; (*Track Delay preset*)
		PTTrack901 : UDINT; (*Track Delay preset*)
		PTTrack011 : UDINT; (*Track Delay preset*)
		PTTrack012 : UDINT; (*Track Delay preset*)
		PTTrack013 : UDINT; (*Track Delay preset*)
		PTTrack101 : UDINT; (*Track Delay preset*)
		PTTrack102 : UDINT; (*Track Delay preset*)
		PTTrack103 : UDINT; (*Track Delay preset*)
		PTTrack104 : UDINT; (*Track Delay preset*)
		PTTrack105 : UDINT; (*Track Delay preset*)
		PTTrack106 : UDINT; (*Track Delay preset*)
		PTTrack107 : UDINT; (*Track Delay preset*)
		PTTrack108 : UDINT; (*Track Delay preset*)
		PTTrack911 : UDINT; (*Track Delay preset*)
		PTTrack912 : UDINT; (*Track Delay preset*)
		PTTrack913 : UDINT; (*Track Delay preset*)
		PTTrack111 : UDINT; (*Track Delay preset*)
		PTTrack112 : UDINT; (*Track Delay preset*)
		PTTrack113 : UDINT; (*Track Delay preset*)
		PTTrack114 : UDINT; (*Track Delay preset*)
		PTTrack115 : UDINT; (*Track Delay preset*)
		PTTrack201 : UDINT; (*Track Delay preset*)
		PTTrack202 : UDINT; (*Track Delay preset*)
		PTTrack203 : UDINT; (*Track Delay preset*)
		PTTrack204 : UDINT; (*Track Delay preset*)
		PTTrack205 : UDINT; (*Track Delay preset*)
		PTTrack206 : UDINT; (*Track Delay preset*)
		PTTrack207 : UDINT; (*Track Delay preset*)
		PTTrack208 : UDINT; (*Track Delay preset*)
		PTTrack921 : UDINT; (*Track Delay preset*)
		PTTrack922 : UDINT; (*Track Delay preset*)
		PTTrack301 : UDINT; (*Track Delay preset*)
		PTTrack302 : UDINT; (*Track Delay preset*)
		PTTrack931 : UDINT; (*Track Delay preset*)
		PTTrack932 : UDINT; (*Track Delay preset*)
		PTTrack401 : UDINT; (*Track Delay preset*)
		PTTrack402 : UDINT; (*Track Delay preset*)
		PTTrack411 : UDINT; (*Track Delay preset*)
		PTTrack412 : UDINT; (*Track Delay preset*)
		PTTrack413 : UDINT; (*Track Delay preset*)
		PTTrack414 : UDINT; (*Track Delay preset*)
		PTTrack501 : UDINT; (*Track Delay preset*)
		PTTrack502 : UDINT; (*Track Delay preset*)
		PTTrack503 : UDINT; (*Track Delay preset*)
		PTTrack504 : UDINT; (*Track Delay preset*)
		PTTrack505 : UDINT; (*Track Delay preset*)
		PTTrack506 : UDINT; (*Track Delay preset*)
		PTTrack507 : UDINT; (*Track Delay preset*)
		PTTrack601 : UDINT; (*Track Delay preset*)
		PTTrack602 : UDINT; (*Track Delay preset*)
		PTTrack603 : UDINT; (*Track Delay preset*)
		PTTrack701 : UDINT; (*Track Delay preset*)
		PTTrack801 : UDINT; (*Track Delay preset*)
		PTTrack802 : UDINT; (*Track Delay preset*)
		PTTrack803 : UDINT; (*Track Delay preset*)
		PTTrack804 : UDINT; (*Track Delay preset*)
		PTTrack805 : UDINT; (*Track Delay preset*)
		PTTrack811 : UDINT; (*Track Delay preset*)
		PTTrack812 : UDINT; (*Track Delay preset*)
		PTTrack821 : UDINT; (*Track Delay preset*)
		PTTrack822 : UDINT; (*Track Delay preset*)
	END_STRUCT;
	VisFlip_typ : 	STRUCT
		Runtime2 : Status_enum := HIDE; (*Runtime display*)
		Runtime4 : Status_enum := HIDE; (*Runtime display*)
		Runtime5 : Status_enum := HIDE; (*Runtime display*)
		Runtime7 : Status_enum := HIDE; (*Runtime display*)
		Runtime9 : Status_enum := HIDE; (*Runtime display*)
		Runtime10 : Status_enum := HIDE; (*Runtime display*)
		Runtime8 : Status_enum := HIDE; (*Runtime display*)
		Runtime6 : Status_enum := HIDE; (*Runtime display*)
		Runtime3 : Status_enum := HIDE; (*Runtime display*)
		Runtime1 : Status_enum := HIDE; (*Runtime display*)
		TextIndex2 : USINT; (*Text Index*)
		TextIndex3 : USINT; (*Text Index*)
		TextIndex4 : USINT; (*Text Index*)
		TextIndex5 : USINT; (*Text Index*)
		TextIndex6 : USINT; (*Text Index*)
		TextIndex7 : USINT; (*Text Index*)
		TextIndex9 : USINT; (*Text Index*)
		TextIndex10 : USINT; (*Text Index*)
		TextIndex11 : USINT; (*Text Index*)
		TextIndex12 : USINT; (*Text Index*)
		TextIndex13 : USINT; (*Text Index*)
		TextIndex14 : USINT; (*Text Index*)
		TextIndex15 : USINT; (*Text Index*)
		TextIndex17 : USINT; (*Text Index*)
		TextIndex18 : USINT; (*Text Index*)
		TextIndex19 : USINT; (*Text Index*)
		TextIndex20 : USINT; (*Text Index*)
		TextIndex16 : USINT; (*Text Index*)
		TextIndex8 : USINT; (*Text Index*)
		TextIndex1 : USINT; (*Text Index*)
		WarnTON1 : TON; (*Warning Delays*)
		WarnTON0 : TON; (*Warning Delays*)
	END_STRUCT;
	VisuControl_enum :
		(
		UNSELECTED := 0,
		SELECTED := 1,
		FOCUS := 4
		);
	X2XModule_typ : 	STRUCT
		OK : BOOL; (*Module status (1 = module present)*)
		SerialNumber : UDINT; (*Serial Number*)
		ID : UINT; (*Module ID*)
		HardwareVariant : UINT; (*Hardware variant*)
		FirmwareVersion : UINT; (*Firmware version*)
		Fuse : BOOL; (*Fuse Status (0 = OK)*)
	END_STRUCT;
	X2X_typ : 	STRUCT
		P1 : BOOL;
		P2 : BOOL;
		P3 : BOOL;
		P4 : BOOL;
		P5 : BOOL;
		P6 : BOOL;
		P7 : BOOL;
		P8 : BOOL;
		P9 : BOOL;
		P10 : BOOL;
		P11 : BOOL;
		P12 : BOOL;
		P13 : BOOL;
		P14 : BOOL;
		P15 : BOOL;
		P16 : BOOL;
	END_STRUCT;
END_TYPE
```

### Global.var - Global variables
```iecst
(********************************************************************
 * COPYRIGHT --
 ********************************************************************
 * File: Global.var
 * Author: NickE
 * Created: April 2, 2015
 ********************************************************************
 * Global variables of project N_Default
 ********************************************************************)
VAR
	AGVInPosition : Input_typ; (*AGV In Position*)
	AGVReceiving : Input_typ; (*AGV Receving Row*)
	AGVReady : Input_typ; (*AGV Operational*)
	AGVReadyToSend : Output_typ; (*Ready to send to AGV*)
	AGVSending : Output_typ; (*Sending to AGV*)
	FurnaceSelect : Mode_typ; (*FALSE = Furnace 1, TRUE = Furnace 2. *)
	Alarm : Alarm_typ; (*Alarm *)
END_VAR
VAR CONSTANT
	AlwaysON : BOOL := TRUE; (*Always On flag*)
END_VAR
VAR RETAIN
	AnalogPerm : ANALOGS_typ;
END_VAR
VAR
	AnalogStore : ANALOGCAPTURE_typ;
END_VAR
VAR RETAIN
	ArmsPerm1 : ArmsPerm_typ; (*Flip up arms retained values*)
	ArmsPerm2 : ArmsPerm_typ; (*Flip up arms retained values*)
END_VAR
VAR
	ArmsTemp1 : FlipUps; (*Flip up arms non retained values*)
	ArmsTemp2 : FlipUps; (*Flip up arms non retained values*)
	Ax1 : Axis_typ; (*Axis 1 variables*)
END_VAR
VAR RETAIN
	Ax1P : AxisPerm_typ; (*Axis 1 permananent variables*)
END_VAR
VAR
	Ax2 : Axis_typ; (*Axis 2 variables*)
END_VAR
VAR RETAIN
	Ax2P : AxisPerm_typ; (*Axis 2 permananent variables*)
END_VAR
VAR
	Ax3 : Axis_typ; (*Axis 3 variables*)
	axis1basic : AxisBasic_typ;
	axis2basic : AxisBasic_typ;
	BatchAtExit : Output_typ; (*Batch ready at exit*)
	BatchMode : BATCHING_enum; (*Batching modes*)
	Belts1 : BeltClear_typ; (*Seamer 1 belts/processing complete*)
	Belts2 : BeltClear_typ; (*Seamer 2 belts/processing complete*)
END_VAR
VAR RETAIN
	CAPT : PTCon_typ; (*Preset times for accumulator conveyor*)
END_VAR
VAR
	CB1 : PLINV_typ; (*Runout conveyor, in line with CC4 & CB2*)
	CB1Test : InvTestFB; (*Test Runout conveyor, in line with CC4 & CB2*)
	CB2 : PLINV_typ; (*Runout conveyor, in line with CB1 & CRB*)
	CB2Test : InvTestFB; (*Test Runout conveyor, in line with CB1 & CRB*)
	CC1 : PLINV_typ; (*Corner conveyor, in line with CS1*)
	CC1Test : InvTestFB; (*Test Corner conveyor, in line with CS1*)
	CC2 : PLINV_typ; (*Corner conveyor, in line with CS2*)
	CC2Test : InvTestFB; (*Test Corner conveyor, in line with CS2*)
	CC3 : PLINV_typ; (*Corner conveyor, in line with CS2*)
	CC3Test : InvTestFB; (*Test Corner conveyor, in line with CS2*)
	CC4 : PLINV_typ; (*Corner conveyor, in line with CB1*)
	CC4Test : InvTestFB; (*Test Corner conveyor, in line with CB1*)
	CL1 : PLINV_typ; (*End loading conveyor, in line with CS1*)
	CL1Test : InvTestFB; (*Test End loading conveyor, in line with CS1*)
	CLB : PLINV_typ; (*Load building conveyor, in line with CRE*)
	CLBTest : InvTestFB; (*Test Load building conveyor, in line with CRE*)
	ClearBatch : Input_typ; (*Clear Batch Button*)
	ClearInv : PLInvOut_typ; (*Reset data at each scan.*)
END_VAR
VAR RETAIN
	CLPT2 : PTCon_typ; (*Preset times for loading conveyor*)
END_VAR
VAR
	Control : ControlFB;
	CRB : PLINV_typ; (*Row building conveyor, in line with CR3*)
	CRBTest : InvTestFB; (*Test Row building conveyor, in line with CR3*)
	CRE : PLINV_typ; (*Row building exit conveyor, in line with CLB*)
	CRETest : InvTestFB; (*Test Row building exit conveyor, in line with CLB*)
	CS1 : PLINV_typ; (*Seamer 1 conveyor, in line with CL1 & CC1*)
	CS1Test : InvTestFB; (*Test Seamer 1 conveyor, in line with CL1 & CC1*)
	CS2 : PLINV_typ; (*Seamer 2 conveyor, in line with CC2 & CR1*)
	CS2Test : InvTestFB; (*Test Seamer 2 conveyor, in line with CC2 & CR1*)
	CV1 : PLINV_typ; (*Seamer 1 vacuum*)
	CV1Test : InvTestFB; (*Test Seamer 1 vacuum*)
	CV2 : PLINV_typ; (*Seamer 2 vacuum*)
	CV2Test : InvTestFB; (*Test Seamer 2 vacuum*)
END_VAR
VAR RETAIN
	Data : Process_typ; (*Runtime data permanent variables*)
END_VAR
VAR
	DataFlow : DataFlow_typ;
	DispStrDecode : Imperialification_typ := (0);
	EMO : EMO_typ; (*EMO Recovery variables*)
	EPLState : EPLState_typ;
	Filstar : Filstar_typ; (*Filstar valve control*)
	FurnReady : Input_typ; (*Furnace ready to accept glass*)
END_VAR
VAR RETAIN
	Grind1 : Grind_typ; (*Grinding data permanent variables*)
	Grind2 : Grind_typ; (*Grinding data permanent variables*)
END_VAR
VAR
	GrindDisp1 : GrindDisp_typ; (*Grinding data display variables*)
	GrindDisp2 : GrindDisp_typ; (*Grinding data display variables*)
	i : INT; (*Array index (Non specific)*)
END_VAR
VAR RETAIN
	InterceptPT : IntervalDelays_typ := (0);
	InvPerms : InvPerms_typ; (*Inverter Permanent Variables*)
END_VAR
VAR
	InvReset : Output_typ; (*Inverter Trip Reset *)
	InvTemps : InvPerms_typ; (*Inverter Variables For visualisation*)
	Laser : Mode_typ; (*Laser variables*)
	LaserBusy : Input_typ; (*Laser Busy (While Marking)*)
	LaserFire : Output_typ; (*Fire Laser Output*)
	LegTest : LegTest_typ;
END_VAR
VAR RETAIN
	LoadPerm : LoadPerm_typ; (*Load building permanent variables*)
END_VAR
VAR
	Loads : Loads_typ;
	LoadTemp : Batch; (*Load building temporary variables*)
	Meterage1 : Display_enum := FB_HIDE;
	Meterage2 : Display_enum := FB_HIDE;
	MeterageReset1 : Measurement_typ := (Reset:=FALSE,Runtime:=FB_HIDE);
	MeterageReset2 : Measurement_typ := (Reset:=FALSE);
	MS1Belt1 : Output_typ; (*Motor Starter 1 - Belt 1 Motor *)
	MS2Belt2 : Output_typ; (*Motor Starter 2 - Belt 2 Motor *)
	MS3Belt3 : Output_typ; (*Motor Starter 3 - Belt 3 Motor *)
	MS4Belt4 : Output_typ; (*Motor Starter 4 - Belt 4 Motor *)
	MS5Belt5 : Output_typ; (*Motor Starter 5 - Belt 5 Motor *)
	MS6Belt6 : Output_typ; (*Motor Starter 6 - Belt 6 Motor *)
	MS7Belt7 : Output_typ; (*Motor Starter 7 - Belt 7 Motor *)
	MS8Belt8 : Output_typ; (*Motor Starter 8 - Belt 8 Motor *)
	MS9Vac1 : Output_typ; (*Motor Starter 9 - Vacuum 1 Pump *)
	MS10Vac2 : Output_typ; (*Motor Starter 10 - Vacuum 2 Pump *)
	MS11Vac3 : Output_typ; (*Motor Starter 11 - Vacuum 3 Pump *)
	MS12Vac4 : Output_typ; (*Motor Starter 12 - Vacuum 4 Pump *)
	MS13Water1 : Output_typ; (*Motor Starter 13 - Water Tank 1 Pump *)
	MS14Water2 : Output_typ; (*Motor Starter 14 - Water Tank 2 Pump *)
	MS19Belt9 : Output_typ; (*Motor Starter 19 - Belt 9 Motor *)
	MS20Belt10 : Output_typ; (*Motor Starter 20 - Belt 10 Motor *)
	MS21Belt11 : Output_typ; (*Motor Starter 21 - Belt 11 Motor *)
	MS22Belt12 : Output_typ; (*Motor Starter 22 - Belt 12 Motor *)
	MS23Vac5 : Output_typ; (*Motor Starter 23 - Extraction Vacuum 5 Pump *)
	MS24Vac6 : Output_typ; (*Motor Starter 24 - Extraction Vacuum 6 Pump *)
	MS25Vac7 : Output_typ; (*Motor Starter 25 - Extraction Vacuum 7 Pump *)
	MS26Vac8 : Output_typ; (*Motor Starter 26 - Extraction Vacuum 8 Pump *)
END_VAR
VAR RETAIN
	NozzlePerm : NozzlePerm_typ := (0);
END_VAR
VAR
	Offline : Mode_typ; (*Manual Batching Loading variables*)
	Pause : Mode_typ; (*Pause mode variables*)
END_VAR
VAR RETAIN
	Perms : Perms_typ; (*Miscellaneous Permanent variables*)
	PresetSeam : PTSeam_typ; (*Auto running timer presets*)
	PresetSys : Preset_typ; (*System timer presets*)
END_VAR
VAR
	ProcessMode : Input_typ; (*Extra process mode input*)
	Reset : Reset_typ; (*Information resets*)
END_VAR
VAR RETAIN
	RowPerm : RowPerm_typ; (*Row building permanent variables*)
END_VAR
VAR
	Rows : Rows_typ;
	RowTemp : Batch; (*Row building temporary variables*)
	S1Photo : Input_typ; (*CL1 Slow Photoelectric Switch*)
	S2Photo : Input_typ; (*CL1 End Photoelectric Switch*)
	S3Photo : Input_typ; (*CS1 Process Photoelectric Switch*)
	S4Photo : Input_typ; (*DG1 Clear Photoelectric Switch*)
	S5Photo : Input_typ; (*Pal2 Clear Photoelectric Switch*)
	S6Photo : Input_typ; (*CC2 Slow Photoelectric Switch*)
	S7Photo : Input_typ; (*CC2 End Photoelectric Switch*)
	S8Photo : Input_typ; (*CS2 Process Photoelectric Switch*)
	S9Photo : Input_typ; (*CS1 Restart Photoelectric Switch*)
	S12Photo : Input_typ; (*CC3 Start Photoelectric Switch*)
	S13Photo : Input_typ; (*CC4 Clear Photoelectric Switch*)
	S14Photo : Input_typ; (*CB1 Stop Photoelectric Switch*)
	S15Photo : Input_typ; (*CB1 Clear Photoelectric Switch*)
	S16Photo : Input_typ; (*CRB Start Photoelectric Switch*)
	S17Photo : Input_typ; (*CRB Stop Photoelectric Switch*)
	S18Photo : Input_typ; (*CRB End Photoelectric Switch*)
	S19Photo : Input_typ; (*CLB Photoelectric Switch*)
	S20Photo : Input_typ; (*Manual Batch Limit Photoelectric Switch*)
	S21Photo : Input_typ; (*CLB End Photoelectric Switch*)
	S30Reed : Input_typ; (*Pallet 1 Down Reed Switch *)
	S31Reed : Input_typ; (*Pallet 1 Up Reed Switch *)
	S32Reed : Input_typ; (*Pallet 2 Down Reed Switch *)
	S33Reed : Input_typ; (*Pallet 2 Up Reed Switch *)
	S34Reed : Input_typ; (*Pallet 3 Down Reed Switch *)
	S35Reed : Input_typ; (*Pallet 3 Up Reed Switch*)
	S36Reed : Input_typ; (*Pallet 4 Down Reed Switch*)
	S37Reed : Input_typ; (*Pallet 4 Up Reed Switch*)
	S38Reed : Input_typ; (*Squaring bar down reed switch*)
	S39Reed : Input_typ; (*Squaring bar up reed switch*)
	S45Foot : Input_typ; (*CL1 Loading Start Footpedal  *)
	S48Foot : Input_typ; (*Manual batch jog footpedal*)
	S49Foot : Input_typ; (*CR2 Clear Footpedal*)
	S50Reed : Input_typ; (*Datum Gate 1 Down Reed Switch *)
	S52Reed : Input_typ; (*Flip Down Arm Up Reed Switch*)
	S53Reed : Input_typ; (*Flip Down Arm Down Reed Switch*)
	S55Lever : Input_typ; (*Line Pause Lever Selector *)
	S56Lever : Input_typ; (*Laser Enabled Lever Selector*)
	S57Lever : Input_typ; (*Offline Loading Lever Selector *)
	S58Lever : Input_typ; (*Manual Batching Lever Selector *)
	S64Float : Input_typ; (*Water Tank 1 Float Switch *)
	S65Float : Input_typ; (*Water Tank 2 Float Switch *)
	S66PB : Input_typ; (*Manual batch complete pushbutton*)
	S80Origin : Input_typ; (*Servo 1 Origin Photoelectric Switch*)
	S81Photo : Input_typ; (*Servo 1 Rev Photoelectric Switch*)
	S82Photo : Input_typ; (*Servo 1 Centre 1 Photoelectric Switch*)
	S83Photo : Input_typ; (*Servo 1 Centre 2 Photoelectric Switch*)
	S84Photo : Input_typ; (*Servo 1 Fwd Photoelectric Switch*)
	S90Origin : Input_typ; (*Servo 2 Origin Photoelectric Switch*)
	S91Photo : Input_typ; (*Servo 2 Rev Photoelectric Switch*)
	S92Photo : Input_typ; (*Servo 2 Centre 1 Photoelectric Switch*)
	S93Photo : Input_typ; (*Servo 2 Centre 2 Photoelectric Switch*)
	S94Photo : Input_typ; (*Servo 2 Fwd Photoelectric Switch*)
	S100Reed : Input_typ; (*Flip Up Arm 1/1 Down Reed Switch*)
	S101Reed : Input_typ; (*Flip Up Arm 1/1 Up Reed Switch*)
	S102Reed : Input_typ; (*Flip Up Arm 1/2 Down Reed Switch*)
	S103Reed : Input_typ; (*Flip Up Arm 1/2 Up Reed Switch*)
	S104Reed : Input_typ; (*Flip Up Arm 2/1 Down Reed Switch*)
	S105Reed : Input_typ; (*Flip Up Arm 2/1 Up Reed Switch*)
	S106Reed : Input_typ; (*Flip Up Arm 2/2 Down Reed Switch*)
	S107Reed : Input_typ; (*Flip Up Arm 2/2 Up Reed Switch*)
	S108Reed : Input_typ; (*Flip Up Arm 3/1 Down Reed Switch*)
	S109Reed : Input_typ; (*Flip Up Arm 3/1 Up Reed Switch*)
	S110Reed : Input_typ; (*Flip Up Arm 3/2 Down Reed Switch*)
	S111Reed : Input_typ; (*Flip Up Arm 3/2 Up Reed Switch*)
	S112Reed : Input_typ; (*Flip Up Arm 4/1 Down Reed Switch*)
	S113Reed : Input_typ; (*Flip Up Arm 4/1 Up Reed Switch*)
	S114Reed : Input_typ; (*Flip Up Arm 4/2 Down Reed Switch*)
	S115Reed : Input_typ; (*Flip Up Arm 4/2 Up Reed Switch*)
	S116Reed : Input_typ; (*Flip Up Arm 5/1 Down Reed Switch*)
	S117Reed : Input_typ; (*Flip Up Arm 5/1 Up Reed Switch*)
	S118Reed : Input_typ; (*Flip Up Arm 5/2 Down Reed Switch*)
	S119Reed : Input_typ; (*Flip Up Arm 5/2 Up Reed Switch*)
	S120Reed : Input_typ; (*Flip Up Arm 6/1 Down Reed Switch*)
	S121Reed : Input_typ; (*Flip Up Arm 6/1 Up Reed Switch*)
	S122Reed : Input_typ; (*Flip Up Arm 6/2 Down Reed Switch*)
	S123Reed : Input_typ; (*Flip Up Arm 6/2 Up Reed Switch*)
	S124Reed : Input_typ; (*Flip Up Arm 7/1 Down Reed Switch*)
	S125Reed : Input_typ; (*Flip Up Arm 7/1 Up Reed Switch*)
	S126Reed : Input_typ; (*Flip Up Arm 7/2 Down Reed Switch*)
	S127Reed : Input_typ; (*Flip Up Arm 7/2 Up Reed Switch*)
	S128Reed : Input_typ; (*Flip Up Arm 8/1 Down Reed Switch*)
	S129Reed : Input_typ; (*Flip Up Arm 8/1 Up Reed Switch*)
	S130Reed : Input_typ; (*Flip Up Arm 8/2 Down Reed Switch*)
	S131Reed : Input_typ; (*Flip Up Arm 8/2 Up Reed Switch*)
	S132Reed : Input_typ; (*Flip Up Arm 9/1 Down Reed Switch*)
	S133Reed : Input_typ; (*Flip Up Arm 9/1 Up Reed Switch*)
	S134Reed : Input_typ; (*Flip Up Arm 9/2 Down Reed Switch*)
	S135Reed : Input_typ; (*Flip Up Arm 9/2 Up Reed Switch*)
	S136Reed : Input_typ; (*Flip Up Arm 10/1 Down Reed Switch*)
	S137Reed : Input_typ; (*Flip Up Arm 10/1 Up Reed Switch*)
	S138Reed : Input_typ; (*Flip Up Arm 10/2 Down Reed Switch*)
	S139Reed : Input_typ; (*Flip Up Arm 10/2 Up Reed Switch*)
END_VAR
VAR RETAIN
	ScalePerm : PLInvScale_typ; (*Conveyor scaling constants*)
END_VAR
VAR
	SeamBlock : ARRAY[0..4] OF BOOL;
	Seamers : SeamersSMProFB; (*Motor and Pump control*)
	SeamersII : SeamersSMProIIFB; (*Motor and Pump control*)
	Seaming : Seamer_typ; (*Seaming variables*)
	Sensor1 : Photo; (*Filter Sensor 1 Input*)
	Sensor2 : Photo; (*Filter Sensor 2 Input*)
	Sensor3 : Photo; (*Filter Sensor 3 Input*)
	Sensor4 : Photo; (*Filter Sensor 4 Input*)
	Sensor5 : Photo; (*Filter Sensor 5 Input*)
	Sensor6 : Photo; (*Filter Sensor 6 Input*)
	Sensor7 : Photo; (*Filter Sensor 7 Input*)
	Sensor8 : Photo; (*Filter Sensor 8 Input*)
	Sensor9 : Photo; (*Filter Sensor 9 Input*)
	Sensor12 : Photo; (*Filter Sensor 12 Input*)
	Sensor13 : Photo; (*Filter Sensor 13 Input*)
	Sensor14 : Photo; (*Filter Sensor 14 Input*)
	Sensor15 : Photo; (*Filter Sensor 15 Input*)
	Sensor16 : Photo; (*Filter Sensor 16 Input*)
	Sensor17 : Photo; (*Filter Sensor 17 Input*)
	Sensor18 : Photo; (*Filter Sensor 18 Input*)
	Sensor19 : Photo; (*Filter Sensor 19 Input*)
	Sensor20 : Photo; (*Filter Sensor 20 Input*)
	Sensor21 : Photo; (*Filter Sensor 21 Input*)
	Servo1NOT : Input_typ; (*Servo 1 Negative Over Travel Limit Switch*)
	Servo1POT : Input_typ; (*Servo 1 Positive Over Travel Limit Switch*)
	Servo2NOT : Input_typ; (*Servo 2 Negative Over Travel Limit Switch*)
	Servo2POT : Input_typ; (*Servo 2 Positive Over Travel Limit Switch*)
	Simulation : Simulation_typ; (*Simulation variables*)
	Sol1Blt1 : Output_typ; (*Solenoid Valve 1 Belt 1 *)
	Sol2Blt2 : Output_typ; (*Solenoid Valve 2 Belt 2 *)
	Sol3Blt3 : Output_typ; (*Solenoid Valve 3 Belt 3*)
	Sol4Blt4 : Output_typ; (*Solenoid Valve 4 Belt 4*)
	Sol5Arm1 : Output_typ; (*Solenoid Valve 5 Flip Up Arm 1*)
	Sol6Arm2 : Output_typ; (*Solenoid Valve 6 Flip Up Arm 2*)
	Sol7Arm3 : Output_typ; (*Solenoid Valve 7 Flip Up Arm 3*)
	Sol8Arm4 : Output_typ; (*Solenoid Valve 8 Flip Up Arm 4*)
	Sol10Blt5 : Output_typ; (*Solenoid Valve 10 Belt 5*)
	Sol11Blt6 : Output_typ; (*Solenoid Valve 11 Belt 6*)
	Sol12Blt7 : Output_typ; (*Solenoid Valve 12 Belt 7*)
	Sol13Blt8 : Output_typ; (*Solenoid Valve 13 Belt 8*)
	Sol14Arm6 : Output_typ; (*Solenoid Valve 14 Flip Up Arm 6*)
	Sol15Arm7 : Output_typ; (*Solenoid Valve 15 Flip Up Arm 7*)
	Sol19Pump : Output_typ; (*Solenoid Valve 19 Scavenge Pump*)
	Sol20DT1 : Output_typ; (*Solenoid Valve 20 Detension 1*)
	Sol21DT2 : Output_typ; (*Solenoid Valve 21 Detension 2*)
	Sol22DT3 : Output_typ; (*Solenoid Valve 22 Detension 3*)
	Sol23DT4 : Output_typ; (*Solenoid Valve 23 Detension 4 *)
	Sol24DG1 : Output_typ; (*Solenoid Valve 24 Datum Gate 1*)
	Sol24DG1B : Output_typ; (*Solenoid Valve 24 Datum Gate 1 B*)
	Sol30Pal1 : Output_typ; (*Solenoid Valve 30 Pallet 1 *)
	Sol31Pal2 : Output_typ; (*Solenoid Valve 31 Pallet 2 *)
	Sol32Pal3 : Output_typ; (*Solenoid Valve 32 Pallet 3*)
	Sol33Pal4 : Output_typ; (*Solenoid Valve 33 Pallet 4*)
	Sol34Pal5 : Output_typ; (*Solenoid Valve 34 Pallet 5*)
	Sol35Laser : Output_typ; (*Solenoid Valve 35 Laser Air Knife*)
	Sol37Spray : Output_typ; (*Solenoid Valve 37 Atomiser Spray*)
	Sol40Datum : Output_typ; (*Solenoid Valve 40 Datum*)
	Sol47Spray : Output_typ; (*Solenoid Valve 47 Atomiser Spray 2*)
	Sol53Recirc : Output_typ; (*Solenoid Valve 53 Recirculation*)
END_VAR
VAR RETAIN
	Speeds : PLInvPerm; (*Conveyor speeds*)
END_VAR
VAR
	Spray1 : NozzleControl; (*Seamer 1 Spray Nozzle*)
	Spray2 : NozzleControl; (*Seamer 2 Spray Nozzle*)
END_VAR
VAR RETAIN
	SysPerm : PermSys_typ; (*Permanent system variables*)
END_VAR
VAR
	SysTemp : TempSys_typ; (*System temporary variables*)
	TestAuto : Input_typ; (*Test Mode Enabled*)
	TestServos : BOOL; (*During Servo Testing*)
	Track001 : TrackBit; (*TRACK FROM S45Foot.In (P) TO S31Reed.In (P)*)
	Track002 : TrackBit; (*TRACK FROM S31Reed.In (P) TO S1Photo.Int (P)*)
	Track003 : TrackBit; (*TRACK FROM S1Photo.Int (P) TO S2Photo.Int (P)*)
	Track004 : TrackBit; (*TRACK FROM S2Photo.Int (P) TO Ax1.SeekFin (P)*)
	Track005 : TrackBit; (*TRACK FROM Ax1.SeekFin (P) TO NOT Tracking00.Blocked (-)*)
	Track011 : TrackBit; (*TRACK FROM S2Photo.Int (P) TO Track011.DelayTON.Q (-)*)
	Track012 : TrackBit; (*TRACK FROM Track011.DelayTON.Q (-) TO LaserBusy.In (N)*)
	Track013 : TrackBit; (*TRACK FROM LaserBusy.In (N) TO NOT Tracking01.Blocked (-)*)
	Track101 : TrackBit; (*TRACK FROM NOT Tracking00.Blocked (-) TO S3Photo.Int (P)*)
	Track102 : TrackBit; (*TRACK FROM S3Photo.Int (P) TO S3Photo.Int (N)*)
	Track103 : TrackBit; (*TRACK FROM S3Photo.Int (N) TO Belts1.Done (P)*)
	Track104 : TrackBit; (*TRACK FROM Belts1.Done (P) TO S4Photo.Int (N)*)
	Track105 : TrackBit; (*TRACK FROM S4Photo.Int (N) TO Track105.DelayTON.Q (P)*)
	Track106 : TrackBit; (*TRACK FROM Track105.DelayTON.Q (P) TO S50Reed.In (P)*)
	Track107 : TrackBit; (*TRACK FROM S50Reed.In (P) TO Track107.DelayTON.Q (P)*)
	Track108 : TrackBit; (*TRACK FROM Track107.DelayTON.Q (P) TO NOT Tracking10.Blocked (-)*)
	Track111 : TrackBit; (*TRACK FROM NOT Tracking10.Blocked (P) TO S32Reed.In (P)*)
	Track112 : TrackBit; (*TRACK FROM S32Reed.In (P) TO S6Photo.Int (P)*)
	Track113 : TrackBit; (*TRACK FROM S6Photo.Int (P) TO S7Photo.Int (P)*)
	Track114 : TrackBit; (*TRACK FROM S7Photo.Int (P) TO Ax2.SeekFin (P)*)
	Track115 : TrackBit; (*TRACK FROM Ax2.SeekFin (P) TO NOT Tracking11.Blocked (-)*)
	Track201 : TrackBit; (*TRACK FROM NOT Tracking11.Blocked (-) TO S8Photo.Int (P)*)
	Track202 : TrackBit; (*TRACK FROM S8Photo.Int (P) TO S8Photo.Int (N)*)
	Track203 : TrackBit; (*TRACK FROM S8Photo.Int (N) TO Belts2.Done (P)*)
	Track204 : TrackBit; (*TRACK FROM Belts2.Done (P) TO S12Photo.Int (N)*)
	Track205 : TrackBit; (*TRACK FROM S12Photo.Int (N) TO Track205.DelayTON.Q (P)*)
	Track206 : TrackBit; (*TRACK FROM Track205.DelayTON.Q (P) TO Track206.DelayTON.Q (P)*)
	Track207 : TrackBit; (*TRACK FROM Track206.DelayTON.Q (P) TO S35Reed.In (P)*)
	Track208 : TrackBit; (*TRACK FROM S35Reed.In (P) TO NOT Tracking20.Blocked (-)*)
	Track301 : TrackBit; (*TRACK FROM NOT Tracking20.Blocked (-) TO S14Photo.Int (P)*)
	Track302 : TrackBit; (*TRACK FROM S14Photo.Int (P) TO NOT Tracking30.Blocked (-)*)
	Track401 : TrackBit; (*TRACK FROM NOT Tracking30.Blocked (-) TO S16Photo.Int (P)*)
	Track402 : TrackBit; (*TRACK FROM S16Photo.Int (P) TO NOT Tracking40.Blocked (-)*)
	Track411 : TrackBit; (*TRACK FROM NOT Tracking40.Blocked (-) TO Track411.DelayTON.Q (P)*)
	Track412 : TrackBit; (*TRACK FROM Track411.DelayTON.Q (P) TO S17Photo.Int (N)*)
	Track413 : TrackBit; (*TRACK FROM S17Photo.Int (N) TO S17Photo.Int (P)*)
	Track414 : TrackBit; (*TRACK FROM S17Photo.Int (P) TO S17Photo.Int (N)*)
	Track501 : TrackBit; (*TRACK FROM S17Photo.Int (N) TO RowTemp.Done (P)*)
	Track502 : TrackBit; (*TRACK FROM RowTemp.Done (P) TO Track502.DelayTON.Q (P)*)
	Track503 : TrackBit; (*TRACK FROM Track502.DelayTON.Q (P) TO S36Reed.In (P)*)
	Track504 : TrackBit; (*TRACK FROM S36Reed.In (P) TO S19Photo.Int (P)*)
	Track505 : TrackBit; (*TRACK FROM S19Photo.Int (P) TO Track505.DelayTON.Q (N)*)
	Track506 : TrackBit; (*TRACK FROM Track505.DelayTON.Q (P) TO S19Photo.Int (N)*)
	Track507 : TrackBit; (*TRACK FROM S19Photo.Int (N) TO Track507.DelayTON.Q (P)*)
	Track511 : TrackBit; (*TRACK FROM S58Lever.Int (P) TO S66PB.In (P)*)
	Track512 : TrackBit; (*TRACK FROM S66PB.In (P) TO S21Photo.In (P)*)
	Track513 : TrackBit; (*TRACK FROM S21Photo.Int (P) TO NOT(Tracking51.Blocked) (-)*)
	Track521 : TrackBit; (*TRACK FROM Track502.DelayTON.Q (P) TO NOT(Tracking52.Blocked) (-)*)
	LengthUnpack : ARRAY[0..15] OF BOOL := [16(FALSE)]; (*Bit array to unpack Row Length*)
	Track522 : TrackBit; (*TRACK FROM NOT(Tracking52.Blocked) (-)  TO Track522.DelayTON.Q (P)*)
	Track601 : TrackBit; (*TRACK FROM Track507.DelayTON.Q(Stop) (P) TO LoadTemp.Done (P)*)
	Track602 : TrackBit; (*TRACK FROM LoadTemp.Done (P) TO S21Photo.Int (P)*)
	Track603 : TrackBit; (*TRACK FROM S21Photo.Int (P) TO NOT(Tracking60.Blocked) (-)*)
	Track701 : TrackBit; (*TRACK FROM NOT(Tracking60.Blocked) (-) TO Track701.DelayTON.Q (P)*)
	Track801 : TrackBit; (*TRACK FROM S18Photo.Int (P) TO S18Photo.Int (N)*)
	Track802 : TrackBit; (*TRACK FROM S18Photo.Int (N) TO Track802.DelayTON.Q (P)*)
	Track803 : TrackBit; (*TRACK FROM Track802.DelayTON.Q (P) TO S36Reed.In (P)*)
	Track804 : TrackBit; (*TRACK FROM S36Reed.In (P) TO S19Photo.Int (P)*)
	Track805 : TrackBit; (*TRACK FROM S19Photo.Int (P) TO S19Photo.Int (N)*)
	Track811 : TrackBit; (*TRACK FROM S19Photo.Int (N) TO S21Photo.Int (P)*)
	Track812 : TrackBit; (*TRACK FROM S21Photo.Int (P) TO NOT(Tracking81.Blocked) (-)*)
	Track821 : TrackBit; (*TRACK FROM NOT(Tracking81.Blocked) (-) TO S21Photo.Int (N)*)
	Track822 : TrackBit; (*TRACK FROM S21Photo.Int (N) TO Track821.DelayTON.Q (P)*)
	Track901 : TrackBit; (*TRACK FROM NOT Tracking00.Blocked (-) TO S2Photo.Int (N)*)
	Track911 : TrackBit; (*TRACK FROM NOT Tracking10.Blocked (-) TO NOT S9Photo.Int (-)*)
	Track912 : TrackBit; (*TRACK FROM NOT S9Photo.Int (-) TO S5Photo.Int (N)*)
	Track921 : TrackBit; (*TRACK FROM NOT Tracking20.Blocked (-) TO Track921.DelayTON.Q (P)*)
	Track922 : TrackBit; (*TRACK FROM Track521.DelayTON.Q (P) TO NOT(S13Photo.Int) (-)*)
	Track931 : TrackBit; (*TRACK FROM NOT Tracking30.Blocked (-) TO S15Photo.Int (N)*)
	Track932 : TrackBit; (*TRACK FROM S15Photo.Int (N) TO Track932.DelayTON.Q (P)*)
	Track941 : TrackBit; (*TRACK FROM NOT Tracking11.Blocked (-) TO S7Photo.Int (N)*)
	TrackClear : TrackBit := (FixedIN:=(Control:=FALSE,ESClearing:=FALSE,EMOStart:=FALSE),RunBlock:=FALSE,SolBlock:=FALSE,Analog:=0,Speed:=0.0,SpeedAnalog:=0.0,SpeedMatchEN:=FALSE,SpeedMatch:=0.0,TimeoutBlock:=FALSE,TimeoutEN:=FALSE,TrackDelayEN:=FALSE,DelayPT:=0,TimeoutACK:=FALSE,DoneIN:=FALSE,Active:=FALSE,Done:=FALSE,Disp:=HIDE,ESDisp:=HIDE,RunOUT:=FALSE,SolOUT:=FALSE,SpeedOUT:=0.0,TimeoutOUT:=FALSE,DelayTON:=(IN:=FALSE),TimeoutACKLatch:=FALSE);
END_VAR
VAR RETAIN
	TrackDelayPT : TrackDelayPT_typ; (*Preset for timeout*)
END_VAR
VAR
	Tracking00 : TrackingSection; (*TRACK BITS Track001 ~ Track005*)
	Tracking01 : TrackingSection; (*TRACK BITS Track011 ~ Track013*)
	Tracking10 : TrackingSection; (*TRACK BITS Track101 ~ Track108*)
	Tracking11 : TrackingSection; (*TRACK BITS Track111 ~ Track115*)
	Tracking20 : TrackingSection; (*TRACK BITS Track201 ~ Track208*)
	Tracking30 : TrackingSection; (*TRACK BITS Track301 ~ Track302*)
	Tracking40 : TrackingSection; (*TRACK BITS Track401 ~ Track402*)
	Tracking41 : TrackingSection; (*TRACK BITS Track411 ~ Track414*)
	Tracking50 : TrackingSection; (*TRACK BITS Track501 ~ Track507*)
	Tracking52 : TrackingSection; (*TRACK BITS Track521 ~ Track522*)
	Tracking51 : TrackingSection; (*TRACK BITS Track511 ~ Track513*)
	Tracking60 : TrackingSection; (*TRACK BITS Track601 ~ Track603*)
	Tracking70 : TrackingSection; (*TRACK BITS Track701 ~ Track603*)
	Tracking80 : TrackingSection; (*TRACK BITS Track801 ~ Track805*)
	Tracking81 : TrackingSection; (*TRACK BITS Track811 ~ Track812*)
	Tracking82 : TrackingSection; (*TRACK BITS Track821 ~ Track822*)
	Tracking90 : TrackingSection; (*TRACK BITS Track901 ~ Track005*)
	Tracking91 : TrackingSection; (*TRACK BITS Track911 ~ Track912*)
	Tracking92 : TrackingSection; (*TRACK BITS Track921 ~ Track922*)
	Tracking93 : TrackingSection; (*TRACK BITS Track931 ~ Track932*)
	Tracking94 : TrackingSection; (*TRACK BITS Track941*)
	Warn : Warnings_typ; (*Timeout variables*)
	Warning : Alarm_typ; (*Warning*)
	WashRun : Input_typ; (*Washer Running  *)
	WashStop : Output_typ; (*Glass running out signal to following equipment*)
	X2X02 : X2X_typ; (*X2X + Station Number*)
	X2X03 : X2X_typ; (*X2X + Station Number*)
	X2X04 : X2X_typ; (*X2X + Station Number*)
	X2X08 : X2X_typ; (*X2X + Station Number*)
	X2X10 : X2X_typ; (*X2X + Station Number*)
	X2X11 : X2X_typ; (*X2X + Station Number*)
	X2X12 : X2X_typ; (*X2X + Station Number*)
	X2X13 : X2X_typ; (*X2X + Station Number*)
	X2X14 : X2X_typ; (*X2X + Station Number*)
	X2X15 : X2X_typ; (*X2X + Station Number*)
	X2X16 : X2X_typ; (*X2X + Station Number*)
	X2X17 : X2X_typ; (*X2X + Station Number*)
	X2X18 : X2X_typ; (*X2X + Station Number*)
	X2X20 : X2X_typ; (*X2X + Station Number*)
	X2X21 : X2X_typ; (*X2X + Station Number*)
	X2X22 : X2X_typ; (*X2X + Station Number*)
	X2XModule : ARRAY[0..30] OF X2XModule_typ; (*X2X Module*)
END_VAR
```

### Package Logical/Libraries - Global libraries

### Library Logical/Libraries/AxisCtrl (IEC, version 0.00.0)

#### AxisCtrl.fun
```iecst
FUNCTION_BLOCK AxisAbsMoveConv
	VAR_INPUT
		Axis	:REFERENCE TO ACP10AXIS_typ;
		Enable	:BOOL;
		AxisMoveAbs	:AxisMoveAbs_typ;
	END_VAR
	VAR_OUTPUT
		Velocity	:REAL;
		Acceleration	:REAL;
		Deceleration	:REAL;
	END_VAR
END_FUNCTION_BLOCK
FUNCTION_BLOCK AxisHomeStatus
	VAR_INPUT
		Enable	:BOOL;
		Clock	:BOOL;
		AxisCtrl	:REFERENCE TO AxisControlAndStatus_typ;
	END_VAR
	VAR_OUTPUT
		HomeStatus	:UINT;
	END_VAR
END_FUNCTION_BLOCK
FUNCTION_BLOCK AxisDriveStatus
	VAR_INPUT
		Axis	:REFERENCE TO ACP10AXIS_typ;
		Enable	:BOOL;
	END_VAR
	VAR_OUTPUT
		RefSw	:BOOL;
		PosSw	:BOOL;
		NegSw	:BOOL;
		Trigger1	:BOOL;
		Trigger2	:BOOL;
		EnableSw	:BOOL;
		HomedOK	:BOOL;
	END_VAR
END_FUNCTION_BLOCK
FUNCTION_BLOCK AxisBrakeStatus
	VAR_INPUT
		Enable	:BOOL;
		StatusPV	:UDINT;
	END_VAR
	VAR_OUTPUT
		RelayOn	:BOOL;
		ElectricalOn	:BOOL;
		MechanicalOpen	:BOOL;
	END_VAR
END_FUNCTION_BLOCK
FUNCTION_BLOCK AxisClearErrorTxt
	VAR_INPUT
		Enable	:BOOL;
		DataAddress	:UDINT;
	END_VAR
	VAR_OUTPUT
		Done	:BOOL;
		Busy	:BOOL;
		Error	:BOOL;
		ErrorID	:UINT;
	END_VAR
END_FUNCTION_BLOCK
FUNCTION_BLOCK AxisFaultStatus
	VAR_INPUT
		Enable	:BOOL;
		Clock	:BOOL;
		AxisCtrl	:REFERENCE TO AxisControlAndStatus_typ;
	END_VAR
	VAR_OUTPUT
		FaultStatus	:UINT;
	END_VAR
END_FUNCTION_BLOCK
FUNCTION_BLOCK AxisCfgToAxisObj
	VAR_INPUT
		Axis	:REFERENCE TO ACP10AXIS_typ;
		Execute	:BOOL;
		AxisConfig	:AxisConfig_typ;
	END_VAR
	VAR_OUTPUT
		Done	:BOOL;
	END_VAR
END_FUNCTION_BLOCK
FUNCTION_BLOCK AxisObjToAxisCfg
	VAR_INPUT
		Axis	:REFERENCE TO ACP10AXIS_typ;
		Execute	:BOOL;
	END_VAR
	VAR_OUTPUT
		Done	:BOOL;
		AxisConfig	:AxisConfig_typ;
	END_VAR
END_FUNCTION_BLOCK
FUNCTION_BLOCK AxisSwitchCfg
	VAR_INPUT
		Axis	:UDINT;
		Execute	:BOOL;
		DeviceName	:STRING[49];
		ChannelName	:STRING[49];
	END_VAR
	VAR_OUTPUT
		Done	:BOOL;
		Busy	:BOOL;
		Error	:BOOL;
		ErrorID	:UINT;
	END_VAR
	VAR
		TempUSINT	:ARRAY[0..19] OF USINT;
		TempUINT	:ARRAY[0..19] OF UINT;
		TempUDINT	:ARRAY[0..19] OF UDINT;
		DataType	:ARRAY[0..19] OF UINT;
		DataAddress	:ARRAY[0..19] OF UDINT;
		ParID	:ARRAY[0..19] OF UINT;
		OffsetCalculated	:BOOL;
		plActionStatus	:UINT;
		BitOffset	:BITOFFSET_typ;
		GetPLOffset_0	:PLACTION_GET_CROSSLINK_INFO_typ;
		ConfigMA3Pos	:CONFIG_MA_CYCLIC_POS_typ;
		MC_BR_WriteParID_0	:MC_BR_WriteParID;
		i	:UINT;
	END_VAR
END_FUNCTION_BLOCK
FUNCTION_BLOCK AxisVelMoveConv
	VAR_INPUT
		Axis	:REFERENCE TO ACP10AXIS_typ;
		Enable	:BOOL;
		AxisMoveVel	:AxisMoveVel_typ;
	END_VAR
	VAR_OUTPUT
		Velocity	:REAL;
		Acceleration	:REAL;
		Deceleration	:REAL;
	END_VAR
END_FUNCTION_BLOCK
```

#### AxisCtrl.typ
```iecst
TYPE
	CONFIG_MA_CYCLIC_POS_typ : STRUCT
		node_number	: UINT ;
		send_parid	: UINT ;
	END_STRUCT;
	BITOFFSET_typ : STRUCT
		node_number	: UINT ;
		offset	: UINT ;
		bits_to_shift	: UINT ;
	END_STRUCT;
	AxisInstrumentation_typ : STRUCT
		StatorCurrent	: REAL ;
		TempModel	: REAL ;
		TempSensor	: REAL ;
		JuctionTemp	: REAL ;
		BleederTemp	: REAL ;
		DCBusVoltage	: REAL ;
		LagError	: REAL ;
		ActPosition	: REAL ;
		ActVelocity	: REAL ;
		ActTorque	: REAL ;
		ActVelocityRPS	: REAL ;
	END_STRUCT;
	AxisControl_typ : STRUCT
		SaveInitPar	: BOOL ;
		Rotary	: BOOL ;
		ControlOn	: BOOL ;
		Reset	: BOOL ;
		HomePermit	: BOOL ;
		Home	: BOOL ;
		MovePermit	: BOOL ;
		StartAbsMove	: ARRAY[0..8] OF BOOL ;
		StartVelMove	: ARRAY[0..1] OF BOOL ;
		StartSyncMove	: BOOL ;
		StopSyncMove	: BOOL ;
		Stop	: BOOL ;
		JogPos	: BOOL ;
		JogNeg	: BOOL ;
		JogStop	: BOOL ;
		SpeedOvR	: REAL ;
		AccDecOvR	: REAL ;
		AckOne	: BOOL ;
		AckAll	: BOOL ;
	END_STRUCT;
	MSG_TEXT_typ : STRUCT
		line1	: STRING[79] ;
		line2	: STRING[79] ;
		line3	: STRING[79] ;
		line4	: STRING[79] ;
	END_STRUCT;
	AxisStatus_typ : STRUCT
		ControllerOn	: BOOL ;
		HomedOK	: BOOL ;
		AbsMoveInPos	: ARRAY[0..8] OF BOOL ;
		VelMoveInVel	: ARRAY[0..1] OF BOOL ;
		Errorstop	: BOOL ;
		Disabled	: BOOL ;
		Stopping	: BOOL ;
		StandStill	: BOOL ;
		DiscreteMotion	: BOOL ;
		ContinuousMotion	: BOOL ;
		SynchronisedMotion	: BOOL ;
		Homing	: BOOL ;
		Moving	: BOOL ;
		JoggingPos	: BOOL ;
		JoggingNeg	: BOOL ;
		FaultAct	: BOOL ;
		NumOfFaults	: UINT ;
		FaultNum	: UINT ;
		FaultTxt	: MSG_TEXT_typ ;
		FaultStatus	: UINT ;
		HomeStatus	: UINT ;
		DriveStatus	: UDINT ;
		BrakeStatus	: UDINT ;
		EnableSw	: BOOL ;
		NegSw	: BOOL ;
		PosSw	: BOOL ;
		RefSw	: BOOL ;
		Trigger1	: BOOL ;
		Trigger2	: BOOL ;
		DriveReady	: BOOL ;
		BrakeRelayOn	: BOOL ;
		BrakeElectricalOn	: BOOL ;
		BrakeMechanicalOpen	: BOOL ;
	END_STRUCT;
	AxisControlAndStatus_typ : STRUCT
		pAxisObject	: UDINT ;
		pAxisCtrl	: UDINT ;
		strAxisInit	: STRING[8] ;
		Node	: USINT ;
		Control	: AxisControl_typ ;
		Status	: AxisStatus_typ ;
		Instrumentation	: AxisInstrumentation_typ ;
	END_STRUCT;
	AxisMoveSync_typ : STRUCT
		CamTable	: STRING[8] ;
		Periodic	: BOOL ;
		MasterOffset	: REAL ;
		SlaveOffset	: REAL ;
		MasterScaling	: REAL ;
		SlaveScaling	: REAL ;
		StartMode	: USINT ;
		MasterParID	: UINT ;
	END_STRUCT;
	AxisMoveVel_typ : STRUCT
		Velocity	: USINT ;
		Acceleration	: USINT ;
		Deceleration	: USINT ;
		Direction	: USINT ;
	END_STRUCT;
	AxisPosition_typ : STRUCT
		Position	: REAL ;
	END_STRUCT;
	AxisMoveAbs_typ : STRUCT
		Position	: REAL ;
		Velocity	: USINT ;
		Acceleration	: USINT ;
		Deceleration	: USINT ;
		Direction	: USINT ;
	END_STRUCT;
	AxisMove_typ : STRUCT
		Position	: ARRAY[0..8] OF AxisPosition_typ ;
		AbsMove	: ARRAY[0..8] OF AxisMoveAbs_typ ;
		VelMove	: ARRAY[0..1] OF AxisMoveVel_typ ;
		SyncMove	: AxisMoveSync_typ ;
	END_STRUCT;
	AxisConfig_typ : STRUCT
		INIT	: BOOL ;
		dig_in_reference	: UINT ;
		dig_in_pos_hw_end	: UINT ;
		dig_in_neg_hw_end	: UINT ;
		dig_in_trigger1	: UINT ;
		dig_in_trigger2	: UINT ;
		encoder_if_count_dir	: USINT ;
		encoder_if_units	: UDINT ;
		encoder_if_rev_motor	: UDINT ;
		limit_v_pos	: REAL ;
		limit_v_neg	: REAL ;
		limit_a1_pos	: REAL ;
		limit_a2_pos	: REAL ;
		limit_a1_neg	: REAL ;
		limit_a2_neg	: REAL ;
		limit_t_jolt	: REAL ;
		limit_t_in_pos	: REAL ;
		limit_pos_sw_end	: DINT ;
		limit_neg_sw_end	: DINT ;
		limit_ds_warning	: REAL ;
		limit_ds_stop	: REAL ;
		limit_a_stop	: REAL ;
		controller_mode	: SINT ;
		position_kv	: REAL ;
		position_tn	: REAL ;
		position_t_predict	: REAL ;
		position_t_total	: REAL ;
		position_p_max	: REAL ;
		position_i_max	: REAL ;
		speed_kv	: REAL ;
		speed_tn	: REAL ;
		speed_t_filter	: REAL ;
		speed_isq_filter1_type	: UINT ;
		speed_isq_filter1_a0	: REAL ;
		speed_isq_filter1_a1	: REAL ;
		speed_isq_filter1_b0	: REAL ;
		speed_isq_filter1_b1	: REAL ;
		speed_isq_filter1_b2	: REAL ;
		speed_isq_filter2_type	: UINT ;
		speed_isq_filter2_a0	: REAL ;
		speed_isq_filter2_a1	: REAL ;
		speed_isq_filter2_b0	: REAL ;
		speed_isq_filter2_b1	: REAL ;
		speed_isq_filter2_b2	: REAL ;
		speed_isq_filter3_type	: UINT ;
		speed_isq_filter3_a0	: REAL ;
		speed_isq_filter3_a1	: REAL ;
		speed_isq_filter3_b0	: REAL ;
		speed_isq_filter3_b1	: REAL ;
		speed_isq_filter3_b2	: REAL ;
		uf_type	: USINT ;
		uf_auto_config	: USINT ;
		uf_u0	: REAL ;
		uf_un	: REAL ;
		uf_fn	: REAL ;
		ff_torque_load	: REAL ;
		ff_torque_pos	: REAL ;
		ff_torque_neg	: REAL ;
		ff_kv_torque	: REAL ;
		ff_inertia	: REAL ;
		ff_t_filter_a	: REAL ;
		stop_decel_ramp	: USINT ;
		stop_controller	: USINT ;
		homing_s	: DINT ;
		homing_v_switch	: REAL ;
		homing_v_trigger	: REAL ;
		homing_a	: REAL ;
		homing_mode	: USINT ;
		homing_edge_sw	: USINT ;
		homing_start_dir	: USINT ;
		homing_trigg_dir	: USINT ;
		homing_ref_pulse	: USINT ;
		homing_tr_s_block	: REAL ;
	END_STRUCT;
END_TYPE
```

#### AxisAbsMoveConv.ab
```automation-basic
FUNCTION_BLOCK AxisAbsMoveConv
	(* Implementation of AxisGoToConv *)

	if (Enable) then
		Velocity = Axis.limit.parameter.v_pos * REAL(AxisMoveAbs.Velocity) * 0.01
		Acceleration = Axis.limit.parameter.a1_pos * REAL(AxisMoveAbs.Acceleration) * 0.01
		Deceleration = Axis.limit.parameter.a2_pos * REAL(AxisMoveAbs.Deceleration) * 0.01
	else
		Velocity = 0.0
		Acceleration = 0.0
		Deceleration = 0.0
	endif
END_FUNCTION_BLOCK
```

#### AxisBrakeStatus.ab
```automation-basic
FUNCTION_BLOCK AxisBrakeStatus
	(*	Bit0: Brake Relay On
			Bit1: Brake Electrical On
			Bit2: Brake Mechanical Open		*)

	if (Enable) then
		RelayOn					=	BIT_TST(StatusPV,1)
		ElectricalOn		= BIT_TST(StatusPV,2)
		MechanicalOpen	= BIT_TST(StatusPV,4)
	else
		RelayOn					= 0
		ElectricalOn		= 0
		MechanicalOpen 	= 0
	endif

END_FUNCTION_BLOCK
```

#### AxisCfgToAxisObj.ab
```automation-basic
FUNCTION_BLOCK AxisCfgToAxisObj
	(* Implementation of AxisCfgToAxisObj *)

	if (Execute) then

		Axis.dig_in.level.reference = AxisConfig.dig_in_reference

		Axis.dig_in.level.pos_hw_end = AxisConfig.dig_in_pos_hw_end
		Axis.dig_in.level.neg_hw_end = AxisConfig.dig_in_neg_hw_end
		Axis.dig_in.level.trigger1 = AxisConfig.dig_in_trigger1
		Axis.dig_in.level.trigger2 = AxisConfig.dig_in_trigger2

		Axis.encoder_if.parameter.count_dir = AxisConfig.encoder_if_count_dir
		Axis.encoder_if.parameter.scaling.load.units = AxisConfig.encoder_if_units
		Axis.encoder_if.parameter.scaling.load.rev_motor = AxisConfig.encoder_if_rev_motor

		Axis.limit.parameter.v_pos = AxisConfig.limit_v_pos
		Axis.limit.parameter.v_neg = AxisConfig.limit_v_neg
		Axis.limit.parameter.a1_pos = AxisConfig.limit_a1_pos
		Axis.limit.parameter.a2_pos = AxisConfig.limit_a2_pos
		Axis.limit.parameter.a1_neg = AxisConfig.limit_a1_neg
		Axis.limit.parameter.a2_neg = AxisConfig.limit_a2_neg
		Axis.limit.parameter.t_jolt = AxisConfig.limit_t_jolt
		Axis.limit.parameter.t_in_pos = AxisConfig.limit_t_in_pos
		Axis.limit.parameter.pos_sw_end = AxisConfig.limit_pos_sw_end
		Axis.limit.parameter.neg_sw_end = AxisConfig.limit_neg_sw_end
		Axis.limit.parameter.ds_warning = AxisConfig.limit_ds_warning
		Axis.limit.parameter.ds_stop = AxisConfig.limit_ds_stop
		Axis.limit.parameter.a_stop = AxisConfig.limit_a_stop

		Axis.controller.mode = AxisConfig.controller_mode
		Axis.controller.position.kv = AxisConfig.position_kv
		Axis.controller.position.tn = AxisConfig.position_tn
		Axis.controller.position.t_predict = AxisConfig.position_t_predict
		Axis.controller.position.t_total = AxisConfig.position_t_total
		Axis.controller.position.p_max = AxisConfig.position_p_max
		Axis.controller.position.i_max = AxisConfig.position_i_max
		Axis.controller.speed.kv = AxisConfig.speed_kv
		Axis.controller.speed.tn = AxisConfig.speed_tn
		Axis.controller.speed.t_filter = AxisConfig.speed_t_filter
		Axis.controller.speed.isq_filter1.type = AxisConfig.speed_isq_filter1_type
		Axis.controller.speed.isq_filter1.a0 = AxisConfig.speed_isq_filter1_a0
		Axis.controller.speed.isq_filter1.a1 = AxisConfig.speed_isq_filter1_a1
		Axis.controller.speed.isq_filter1.b0 = AxisConfig.speed_isq_filter1_b0
		Axis.controller.speed.isq_filter1.b1 = AxisConfig.speed_isq_filter1_b1
		Axis.controller.speed.isq_filter1.b2 = AxisConfig.speed_isq_filter1_b2
		Axis.controller.speed.isq_filter2.type = AxisConfig.speed_isq_filter2_type
		Axis.controller.speed.isq_filter2.a0 = AxisConfig.speed_isq_filter2_a0
		Axis.controller.speed.isq_filter2.a1 = AxisConfig.speed_isq_filter2_a1
		Axis.controller.speed.isq_filter2.b0 = AxisConfig.speed_isq_filter2_b0
		Axis.controller.speed.isq_filter2.b1 = AxisConfig.speed_isq_filter2_b1
		Axis.controller.speed.isq_filter2.b2 = AxisConfig.speed_isq_filter2_b2
		Axis.controller.speed.isq_filter3.type = AxisConfig.speed_isq_filter3_type
		Axis.controller.speed.isq_filter3.a0 = AxisConfig.speed_isq_filter3_a0
		Axis.controller.speed.isq_filter3.a1 = AxisConfig.speed_isq_filter3_a1
		Axis.controller.speed.isq_filter3.b0 = AxisConfig.speed_isq_filter3_b0
		Axis.controller.speed.isq_filter3.b1 = AxisConfig.speed_isq_filter3_b1
		Axis.controller.speed.isq_filter3.b2 = AxisConfig.speed_isq_filter3_b2
		Axis.controller.uf.type = AxisConfig.uf_type
		Axis.controller.uf.auto_config = AxisConfig.uf_auto_config
		Axis.controller.uf.u0 = AxisConfig.uf_u0
		Axis.controller.uf.un = AxisConfig.uf_un
		Axis.controller.uf.fn = AxisConfig.uf_fn
		Axis.controller.ff.torque_load = AxisConfig.ff_torque_load
		Axis.controller.ff.torque_pos = AxisConfig.ff_torque_pos
		Axis.controller.ff.torque_neg = AxisConfig.ff_torque_neg
		Axis.controller.ff.kv_torque = AxisConfig.ff_kv_torque
		Axis.controller.ff.inertia = AxisConfig.ff_inertia

		Axis.move.stop.parameter[0].decel_ramp = AxisConfig.stop_decel_ramp
		Axis.move.stop.parameter[0].controller = AxisConfig.stop_controller

		Axis.move.homing.parameter.s = AxisConfig.homing_s
		Axis.move.homing.parameter.v_switch = AxisConfig.homing_v_switch
		Axis.move.homing.parameter.v_trigger = AxisConfig.homing_v_trigger
		Axis.move.homing.parameter.a = AxisConfig.homing_a
		Axis.move.homing.parameter.mode = AxisConfig.homing_mode
		Axis.move.homing.parameter.edge_sw = AxisConfig.homing_edge_sw
		Axis.move.homing.parameter.start_dir = AxisConfig.homing_start_dir
		Axis.move.homing.parameter.trigg_dir = AxisConfig.homing_trigg_dir
		Axis.move.homing.parameter.ref_pulse = AxisConfig.homing_ref_pulse
		Axis.move.homing.parameter.tr_s_block = AxisConfig.homing_tr_s_block

		Done = true

	else

		Done = false

	endif
END_FUNCTION_BLOCK
```

#### AxisClearErrorTxt.ab
```automation-basic
FUNCTION_BLOCK AxisClearErrorTxt
	(* Implementation of AxisClearError *)

	if (Enable) then
		Busy = True		; Future
		Done = False	; Future
		Error = False	; Future
		ErrorID = 0		; Future
		memset(DataAddress,0,320)
		Busy = False
		Done = True
	else
		Busy = False
		Done = False
		Error = False
		ErrorID = 0
	endif

END_FUNCTION_BLOCK
```

#### AxisDriveStatus.ab
```automation-basic
FUNCTION_BLOCK AxisDriveStatus
	; Decode drive status.

	if (Enable) then
		RefSw 					=	BOOL(Axis.dig_in.status.reference)
		PosSw 					= BOOL(Axis.dig_in.status.pos_hw_end)
		NegSw 					= BOOL(Axis.dig_in.status.neg_hw_end)
		Trigger1 				= BOOL(Axis.dig_in.status.trigger1)
		Trigger2 				= BOOL(Axis.dig_in.status.trigger2)
		EnableSw 				= BOOL(Axis.dig_in.status.enable)
		HomedOK					= BOOL(Axis.move.homing.status.ok)
	else
		RefSw 					= 0
		PosSw 					= 0
		NegSw 					= 0
		Trigger1 				= 0
		Trigger2 				= 0
		EnableSw 				= 0
		HomedOK   			= 0
	endif

END_FUNCTION_BLOCK
```

#### AxisFaultStatus.ab
```automation-basic
FUNCTION_BLOCK AxisFaultStatus
	(* Implementation of AxisFaultStatus *)

	if (Enable) then
		if (AxisCtrl.Status.FaultAct) AND (Clock) then
			AxisCtrl.Status.FaultStatus = 51
		else
			AxisCtrl.Status.FaultStatus = 7
		endif
	else
		AxisCtrl.Status.FaultStatus = 0
	endif

	FaultStatus = AxisCtrl.Status.FaultStatus

END_FUNCTION_BLOCK
```

#### AxisHomeStatus.ab
```automation-basic
FUNCTION_BLOCK AxisHomeStatus
	(* Implementation of AxisHomeStatus *)

	if (Enable) then
		if NOT(AxisCtrl.Status.ControllerOn) then
			AxisCtrl.Status.HomeStatus = 8
		else if NOT(AxisCtrl.Status.HomedOK) then
			AxisCtrl.Status.HomeStatus = 51
		else if (AxisCtrl.Status.Homing) AND (Clock) then
			AxisCtrl.Status.HomeStatus = 46
		else if (AxisCtrl.Status.Homing) AND NOT(Clock) then
			AxisCtrl.Status.HomeStatus = 7
		else if (AxisCtrl.Status.HomedOK) then
			AxisCtrl.Status.HomeStatus = 221
		endif
	else
		AxisCtrl.Status.HomeStatus = 0
	endif

	HomeStatus = AxisCtrl.Status.HomeStatus

END_FUNCTION_BLOCK
```

#### AxisObjToAxisCfg.ab
```automation-basic
FUNCTION_BLOCK AxisObjToAxisCfg
	(* Implementation of AxisObjtoAxisCfg *)

	if (Execute) then

		AxisConfig.dig_in_reference = Axis.dig_in.level.reference
		AxisConfig.dig_in_pos_hw_end = Axis.dig_in.level.pos_hw_end
		AxisConfig.dig_in_neg_hw_end = Axis.dig_in.level.neg_hw_end
		AxisConfig.dig_in_trigger1 = Axis.dig_in.level.trigger1
		AxisConfig.dig_in_trigger2 = Axis.dig_in.level.trigger2

		AxisConfig.encoder_if_count_dir = Axis.encoder_if.parameter.count_dir
		AxisConfig.encoder_if_units = Axis.encoder_if.parameter.scaling.load.units
		AxisConfig.encoder_if_rev_motor = Axis.encoder_if.parameter.scaling.load.rev_motor

		AxisConfig.limit_v_pos = Axis.limit.parameter.v_pos
		AxisConfig.limit_v_neg = Axis.limit.parameter.v_neg
		AxisConfig.limit_a1_pos = Axis.limit.parameter.a1_pos
		AxisConfig.limit_a2_pos = Axis.limit.parameter.a2_pos
		AxisConfig.limit_a1_neg = Axis.limit.parameter.a1_neg
		AxisConfig.limit_a2_neg = Axis.limit.parameter.a2_neg
		AxisConfig.limit_t_jolt = Axis.limit.parameter.t_jolt
		AxisConfig.limit_t_in_pos = Axis.limit.parameter.t_in_pos
		AxisConfig.limit_pos_sw_end = Axis.limit.parameter.pos_sw_end
		AxisConfig.limit_neg_sw_end = Axis.limit.parameter.neg_sw_end
		AxisConfig.limit_ds_warning = Axis.limit.parameter.ds_warning
		AxisConfig.limit_ds_stop = Axis.limit.parameter.ds_stop
		AxisConfig.limit_a_stop = Axis.limit.parameter.a_stop

		AxisConfig.controller_mode = Axis.controller.mode
		AxisConfig.position_kv = Axis.controller.position.kv
		AxisConfig.position_tn = Axis.controller.position.tn
		AxisConfig.position_t_predict = Axis.controller.position.t_predict
		AxisConfig.position_t_total = Axis.controller.position.t_total
		AxisConfig.position_p_max = Axis.controller.position.p_max
		AxisConfig.position_i_max = Axis.controller.position.i_max
		AxisConfig.speed_kv = Axis.controller.speed.kv
		AxisConfig.speed_tn = Axis.controller.speed.tn
		AxisConfig.speed_t_filter = Axis.controller.speed.t_filter
		AxisConfig.speed_isq_filter1_type = Axis.controller.speed.isq_filter1.type
		AxisConfig.speed_isq_filter1_a0 = Axis.controller.speed.isq_filter1.a0
		AxisConfig.speed_isq_filter1_a1 = Axis.controller.speed.isq_filter1.a1
		AxisConfig.speed_isq_filter1_b0 = Axis.controller.speed.isq_filter1.b0
		AxisConfig.speed_isq_filter1_b1 = Axis.controller.speed.isq_filter1.b1
		AxisConfig.speed_isq_filter1_b2 = Axis.controller.speed.isq_filter1.b2
		AxisConfig.speed_isq_filter2_type = Axis.controller.speed.isq_filter2.type
		AxisConfig.speed_isq_filter2_a0 = Axis.controller.speed.isq_filter2.a0
		AxisConfig.speed_isq_filter2_a1 = Axis.controller.speed.isq_filter2.a1
		AxisConfig.speed_isq_filter2_b0 = Axis.controller.speed.isq_filter2.b0
		AxisConfig.speed_isq_filter2_b1 = Axis.controller.speed.isq_filter2.b1
		AxisConfig.speed_isq_filter2_b2 = Axis.controller.speed.isq_filter2.b2
		AxisConfig.speed_isq_filter3_type = Axis.controller.speed.isq_filter3.type
		AxisConfig.speed_isq_filter3_a0 = Axis.controller.speed.isq_filter3.a0
		AxisConfig.speed_isq_filter3_a1 = Axis.controller.speed.isq_filter3.a1
		AxisConfig.speed_isq_filter3_b0 = Axis.controller.speed.isq_filter3.b0
		AxisConfig.speed_isq_filter3_b1 = Axis.controller.speed.isq_filter3.b1
		AxisConfig.speed_isq_filter3_b2 = Axis.controller.speed.isq_filter3.b2
		AxisConfig.uf_type = Axis.controller.uf.type
		AxisConfig.uf_auto_config = Axis.controller.uf.auto_config
		AxisConfig.uf_u0 = Axis.controller.uf.u0
		AxisConfig.uf_un = Axis.controller.uf.un
		AxisConfig.uf_fn = Axis.controller.uf.fn
		AxisConfig.ff_torque_load = Axis.controller.ff.torque_load
		AxisConfig.ff_torque_pos = Axis.controller.ff.torque_pos
		AxisConfig.ff_torque_neg = Axis.controller.ff.torque_neg
		AxisConfig.ff_kv_torque = Axis.controller.ff.kv_torque
		AxisConfig.ff_inertia = Axis.controller.ff.inertia

		AxisConfig.stop_decel_ramp = Axis.move.stop.parameter[0].decel_ramp
		AxisConfig.stop_controller = Axis.move.stop.parameter[0].controller

		AxisConfig.homing_s = Axis.move.homing.parameter.s
		AxisConfig.homing_v_switch = Axis.move.homing.parameter.v_switch
		AxisConfig.homing_v_trigger = Axis.move.homing.parameter.v_trigger
		AxisConfig.homing_a = Axis.move.homing.parameter.a
		AxisConfig.homing_mode = Axis.move.homing.parameter.mode
		AxisConfig.homing_edge_sw = Axis.move.homing.parameter.edge_sw
		AxisConfig.homing_start_dir = Axis.move.homing.parameter.start_dir
		AxisConfig.homing_trigg_dir = Axis.move.homing.parameter.trigg_dir
		AxisConfig.homing_ref_pulse = Axis.move.homing.parameter.ref_pulse
		AxisConfig.homing_tr_s_block = Axis.move.homing.parameter.tr_s_block

		Done = true

	else

		Done = false

	endif

END_FUNCTION_BLOCK
```

#### AxisSwitchCfg.ab
```automation-basic
FUNCTION_BLOCK AxisSwitchCfg
	(* Implementation of AxisSwitchCfg *)

	if (Execute) then

		GetPLOffset_0.DeviceName = ADR(DeviceName)
		GetPLOffset_0.ChannelName = ADR(ChannelName)

		if ((Axis <> 0) AND NOT(OffsetCalculated)) then

			plActionStatus = plAction(0, plACTION_GET_CROSSLINK_INFO, adr(GetPLOffset_0), sizeof(GetPLOffset_0))

			if (plActionStatus = 0) then
				BitOffset.offset = (GetPLOffset_0.Offset / 32) * 32
				BitOffset.bits_to_shift = GetPLOffset_0.Offset mod 32
				BitOffset.node_number = GetPLOffset_0.NodeId
				OffsetCalculated = TRUE

				; PAR ID Data to be written
				; 0
				TempUINT[0] = ACP10PAR_BIT_MODE + 0
				ParID[0] = ACP10PAR_FUNCTION_BLOCK_CREATE
				DataAddress[0]= ADR(TempUINT[0])
				DataType[0]= ncPAR_TYP_UINT
				; 1
				TempUINT[1] = ACP10PAR_ARITH_MODE + 0
				ParID[1]= ACP10PAR_FUNCTION_BLOCK_CREATE
				DataAddress[1]= ADR(TempUINT[1])
				DataType[1] = ncPAR_TYP_UINT
				; 2
				TempUDINT[2] = 1
				ParID[2] = ACP10PAR_BIT_A1 + 0
				DataAddress[2] = ADR(TempUDINT[2])
				DataType[2]	= ncPAR_TYP_UDINT
				; 3
				TempUDINT[3] = 1
				ParID[3] = ACP10PAR_BIT_A2 + 0
				DataAddress[3] = ADR(TempUDINT[3])
				DataType[3] = ncPAR_TYP_UDINT
				; 4
				TempUDINT[4] = 1
				ParID[4] = ACP10PAR_BIT_A3 + 0
				DataAddress[4] = ADR(TempUDINT[4])
				DataType[4] = ncPAR_TYP_UDINT
				; 5
				TempUINT[5] = ACP10PAR_MA3_CYCLIC_POS
				ParID[5] = ACP10PAR_BIT_IN1_PARID + 0
				DataAddress[5] = ADR(TempUINT[5])
				DataType[5] = ncPAR_TYP_UINT
				; 6
				TempUINT[6] = ACP10PAR_MA3_CYCLIC_POS
				ParID[6] = ACP10PAR_BIT_IN2_PARID + 0
				DataAddress[6] = ADR(TempUINT[6])
				DataType[6] = ncPAR_TYP_UINT
				; 7
				TempUINT[7] = ACP10PAR_MA3_CYCLIC_POS
				ParID[7] = ACP10PAR_BIT_IN3_PARID + 0
				DataAddress[7] = ADR(TempUINT[7])
				DataType[7] = ncPAR_TYP_UINT
				; 8
				TempUINT[8] = 10
				ParID[8] = ACP10PAR_BIT_MODE + 0
				DataAddress[8] = ADR(TempUINT[8])
				DataType[8] = ncPAR_TYP_UINT
				; 9
				TempUINT[9] = ACP10PAR_BIT_VALUE1 + 0
				ParID[9] = ACP10PAR_POS_LIMIT_SWITCH_PARID
				DataAddress[9] = ADR(TempUINT[9])
				DataType[9] = ncPAR_TYP_UINT
				; 10
				TempUINT[10] = ACP10PAR_BIT_VALUE2 + 0
				ParID[10] = ACP10PAR_NEG_LIMIT_SWITCH_PARID
				DataAddress[10] = ADR(TempUINT[10])
				DataType[10] = ncPAR_TYP_UINT
				; 11
				TempUINT[11] = ACP10PAR_BIT_VALUE3 + 0
				ParID[11] = ACP10PAR_REFERENCE_SWITCH_PARID
				DataAddress[11] = ADR(TempUINT[11])
				DataType[11] = ncPAR_TYP_UINT
				; 12
				TempUSINT[12] = 0
				ParID[12] = ACP10PAR_MA3_CYCLIC_IPL_MODE
				DataAddress[12] = ADR(TempUSINT[12])
				DataType[12] = ncPAR_TYP_USINT
				; 13
				TempUINT[13] = BitOffset.offset
				ParID[13] = ACP10PAR_CYCLIC_DP_DATA_OFFSET
				DataAddress[13] = ADR(TempUINT[13])
				DataType[13] = ncPAR_TYP_UINT
				; 14
				ConfigMA3Pos.node_number = BitOffset.node_number
				ConfigMA3Pos.send_parid = ACP10PAR_CYCLIC_DP_DATA_OFFSET
				ParID[14] = ACP10PAR_CONFIG_MA3_CYCLIC_POS
				DataAddress[14] = ADR(ConfigMA3Pos)
				DataType[14] = ncPAR_TYP_VOID
				; 15
				TempUINT[15] = 7
				ParID[15] = ACP10PAR_CYCLIC_DP_DATA_TYPE
				DataAddress[15] = ADR(TempUINT[15])
				DataType[15] = ncPAR_TYP_VOID
				; 16
				TempUDINT[16] = BitOffset.bits_to_shift
				ParID[16] = ACP10PAR_BIT_B1+0
				DataAddress[16] = ADR(TempUDINT[16])
				DataType[16] = ncPAR_TYP_UDINT
				; 17
				TempUDINT[17] = BitOffset.bits_to_shift+1
				ParID[17]	= ACP10PAR_BIT_B2+0
				DataAddress[17] = ADR(TempUDINT[17])
				DataType[17] = ncPAR_TYP_UDINT
				; 18
				TempUDINT[18] = BitOffset.bits_to_shift+2
				ParID[18] = ACP10PAR_BIT_B3+0
				DataAddress[18] = ADR(TempUDINT[18])
				DataType[18] = ncPAR_TYP_UDINT

			else
				OffsetCalculated = FALSE
			endif

		endif

		if (OffsetCalculated) AND NOT(Done) AND (Error = FALSE) then

			MC_BR_WriteParID_0.Axis = Axis
			MC_BR_WriteParID_0.Execute = TRUE
			MC_BR_WriteParID_0.ParID = ParID[i]
			MC_BR_WriteParID_0.DataAddress = DataAddress[i]
			MC_BR_WriteParID_0.DataType	= DataType[i]

			MC_BR_WriteParID_0 FUB MC_BR_WriteParID()

			if (MC_BR_WriteParID_0.ErrorID <> 0) then
				Error = TRUE
				ErrorID = MC_BR_WriteParID_0.ErrorID
			endif

			if (MC_BR_WriteParID_0.Done) AND NOT(MC_BR_WriteParID_0.Busy) then
				if (i = 18) then
					i = 0
					Done = TRUE
					Busy = FALSE
				else
					MC_BR_WriteParID_0.Execute = FALSE
					MC_BR_WriteParID_0 FUB MC_BR_WriteParID()
					i = i + 1
					Busy = TRUE
				endif
			endif
		else

			MC_BR_WriteParID_0.Execute = FALSE
			MC_BR_WriteParID_0 FUB MC_BR_WriteParID()

		endif

	else

		i = 0
		OffsetCalculated = FALSE
		Done = FALSE
		Error = FALSE
		ErrorID = 0

	endif

END_FUNCTION_BLOCK
```

#### AxisVelMoveConv.ab
```automation-basic
FUNCTION_BLOCK AxisVelMoveConv
	(* Implementation of AxisVelMoveConv *)

	if (Enable) then
		Velocity = Axis.limit.parameter.v_pos * REAL(AxisMoveVel.Velocity) * 0.01
		Acceleration = Axis.limit.parameter.a1_pos * REAL(AxisMoveVel.Acceleration) * 0.01
		Deceleration = Axis.limit.parameter.a2_pos * REAL(AxisMoveVel.Deceleration) * 0.01
	else
		Velocity = 0.0
		Acceleration = 0.0
		Deceleration = 0.0
	endif

END_FUNCTION_BLOCK
```

### Library Logical/Libraries/IecCheck (IEC) - A library implementing IEC check functions

#### IecCheck.fun - Exported functions and function blocks
```iecst
(********************************************************************
 * COPYRIGHT --
 ********************************************************************
 * Library: IecCheck
 * File: IecCheck.fun
 * Author: NickE
 * Created: July 12, 2011
 ********************************************************************
 * Functions and function blocks of library IecCheck
 ********************************************************************)

FUNCTION CheckDivDWord : UDINT (* Check divisor for DINT and UDINT division *)
	VAR_INPUT
		divisor : UDINT;
	END_VAR
END_FUNCTION

FUNCTION CheckDivWord : UINT (* Check divisor for INT and UINT division *)
	VAR_INPUT
		divisor : UINT;
	END_VAR
END_FUNCTION

FUNCTION CheckDivByte : USINT (* Check divisor for SINT and USINT division *)
	VAR_INPUT
		divisor : USINT;
	END_VAR
END_FUNCTION

FUNCTION CheckDivReal : REAL (* Check divisor for REAL division *)
	VAR_INPUT
		divisor : REAL;
	END_VAR
END_FUNCTION

FUNCTION CheckDivLReal : LREAL (* Check divisor for LREAL division, not available for SG3 and SGC *)
	VAR_INPUT
		divisor : LREAL;
	END_VAR
END_FUNCTION

FUNCTION CheckBounds : DINT (* Check range for array access *)
	VAR_INPUT
		index : DINT;
		lower : DINT;
		upper : DINT;
	END_VAR
END_FUNCTION

FUNCTION CheckRange : DINT (* Check range for enumeration *)
	VAR_INPUT
		value : DINT;
		lower : DINT;
		upper : DINT;
	END_VAR
END_FUNCTION

FUNCTION CheckReadAccess : UDINT (* Check address when reading dynamic variables *)
	VAR_INPUT
		address : UDINT;
	END_VAR
END_FUNCTION

FUNCTION CheckWriteAccess : UDINT (* Check address when writing dynamic variables *)
	VAR_INPUT
		address : UDINT;
	END_VAR
END_FUNCTION
```
